C03664=1140.548,355.302,-81.415,-176.440,9.444,148.890
C03665=1140.545,355.549,-81.451,-176.437,9.448,148.890
C03666=1140.541,355.796,-81.486,-176.435,9.451,148.890
C03667=1140.537,356.044,-81.521,-176.433,9.456,148.891
C03668=1140.533,356.292,-81.556,-176.430,9.460,148.891
C03669=1140.529,356.539,-81.592,-176.427,9.464,148.891
C03670=1140.525,356.787,-81.627,-176.425,9.467,148.892
C03671=1140.522,357.034,-81.661,-176.422,9.472,148.892
C03672=1140.518,357.281,-81.697,-176.420,9.476,148.893
C03673=1140.514,357.529,-81.731,-176.417,9.479,148.893
C03674=1140.510,357.776,-81.767,-176.415,9.484,148.893
C03675=1140.506,358.024,-81.803,-176.412,9.488,148.894
C03676=1140.502,358.272,-81.837,-176.409,9.492,148.894
C03677=1140.498,358.519,-81.873,-176.407,9.497,148.894
C03678=1140.494,358.766,-81.908,-176.405,9.500,148.895
C03679=1140.491,359.014,-81.944,-176.402,9.504,148.895
C03680=1140.486,359.262,-81.980,-176.400,9.509,148.896
C03681=1140.482,359.509,-82.014,-176.397,9.513,148.896
C03682=1140.478,359.756,-82.050,-176.395,9.516,148.896
C03683=1140.474,360.004,-82.085,-176.392,9.521,148.897
C03684=1140.471,360.251,-82.121,-176.389,9.525,148.897
C03685=1140.466,360.498,-82.156,-176.387,9.529,148.897
C03686=1140.463,360.746,-82.192,-176.384,9.534,148.898
C03687=1140.459,360.993,-82.227,-176.381,9.538,148.898
C03688=1140.455,361.241,-82.263,-176.379,9.541,148.899
C03689=1140.452,361.488,-82.298,-176.377,9.546,148.899
C03690=1140.447,361.735,-82.333,-176.374,9.550,148.899
C03691=1140.443,361.983,-82.370,-176.371,9.554,148.900
C03692=1140.439,362.230,-82.405,-176.369,9.558,148.900
C03693=1140.436,362.478,-82.441,-176.366,9.563,148.900
C03694=1140.432,362.725,-82.476,-176.364,9.567,148.901
C03695=1140.428,362.973,-82.512,-176.361,9.571,148.901
C03696=1140.425,363.220,-82.547,-176.358,9.575,148.902
C03697=1140.420,363.467,-82.583,-176.356,9.579,148.902
C03698=1140.416,363.715,-82.619,-176.354,9.583,148.902
C03699=1140.412,363.962,-82.654,-176.351,9.587,148.903
C03700=1140.409,364.210,-82.690,-176.348,9.592,148.903
C03701=1140.405,364.457,-82.725,-176.346,9.596,148.904
C03702=1140.400,364.741,-82.767,-176.342,9.601,148.904
C03703=1140.396,365.025,-82.808,-176.340,9.605,148.904
C03704=1140.392,365.309,-82.849,-176.337,9.611,148.905
C03705=1140.387,365.593,-82.890,-176.333,9.616,148.905
C03706=1140.383,365.840,-82.926,-176.331,9.620,148.906
C03707=1140.380,366.087,-82.962,-176.328,9.624,148.906
C03708=1140.375,366.335,-82.998,-176.325,9.629,148.907
C03709=1140.371,366.582,-83.034,-176.323,9.633,148.907
C03710=1140.368,366.830,-83.069,-176.320,9.637,148.907
C03711=1140.364,367.077,-83.106,-176.318,9.642,148.908
C03712=1140.360,367.324,-83.141,-176.315,9.646,148.908
C03713=1140.356,367.572,-83.177,-176.312,9.650,148.909
C03714=1140.352,367.819,-83.214,-176.310,9.654,148.909
C03715=1140.349,368.066,-83.249,-176.307,9.658,148.909
C03716=1140.345,368.314,-83.285,-176.304,9.663,148.910
C03717=1140.341,368.561,-83.322,-176.302,9.667,148.910
C03718=1140.337,368.809,-83.357,-176.299,9.671,148.910
C03719=1140.333,369.056,-83.394,-176.296,9.676,148.911
C03720=1140.329,369.303,-83.430,-176.294,9.680,148.911
C03721=1140.325,369.550,-83.467,-176.291,9.684,148.912
C03722=1140.322,369.798,-83.502,-176.288,9.688,148.912
C03723=1140.318,370.045,-83.539,-176.286,9.692,148.913
C03724=1140.314,370.293,-83.575,-176.284,9.696,148.913
C03725=1140.311,370.540,-83.611,-176.281,9.700,148.913
C03726=1140.306,370.787,-83.647,-176.278,9.705,148.914
C03727=1140.303,371.034,-83.683,-176.276,9.709,148.914
C03728=1140.298,371.282,-83.719,-176.273,9.714,148.915
C03729=1140.295,371.529,-83.756,-176.270,9.718,148.915
C03730=1140.291,371.776,-83.793,-176.268,9.722,148.915
C03731=1140.287,372.024,-83.829,-176.265,9.726,148.916
C03732=1140.283,372.271,-83.865,-176.263,9.731,148.916
C03733=1140.279,372.518,-83.902,-176.260,9.735,148.917
C03734=1140.275,372.766,-83.937,-176.257,9.739,148.917
C03735=1140.271,373.013,-83.974,-176.255,9.744,148.918
C03736=1140.268,373.260,-84.010,-176.253,9.747,148.918
C03737=1140.264,373.508,-84.047,-176.250,9.752,148.918
C03738=1140.260,373.755,-84.084,-176.248,9.756,148.919
C03739=1140.257,374.002,-84.120,-176.245,9.760,148.919
C03740=1140.253,374.249,-84.157,-176.243,9.765,148.920
C03741=1140.249,374.497,-84.193,-176.240,9.768,148.920
C03742=1140.245,374.744,-84.229,-176.238,9.772,148.921
C03743=1140.241,374.991,-84.266,-176.235,9.777,148.921
C03744=1140.237,375.238,-84.302,-176.233,9.781,148.921
C03745=1140.233,375.485,-84.339,-176.231,9.785,148.922
C03746=1140.230,375.734,-84.376,-176.228,9.789,148.922
C03747=1140.226,375.981,-84.412,-176.227,9.793,148.923
C03748=1140.222,376.228,-84.449,-176.224,9.797,148.923
C03749=1140.218,376.475,-84.486,-176.221,9.801,148.924
C03750=1140.215,376.722,-84.522,-176.220,9.805,148.924
C03751=1140.211,376.969,-84.559,-176.217,9.809,148.925
C03752=1140.207,377.217,-84.596,-176.216,9.813,148.925
C03753=1140.203,377.464,-84.633,-176.213,9.818,148.926
C03754=1140.200,377.711,-84.669,-176.211,9.821,148.926
C03755=1140.196,377.958,-84.706,-176.209,9.825,148.926
C03756=1140.191,378.205,-84.743,-176.207,9.829,148.927
C03757=1140.187,378.453,-84.780,-176.205,9.833,148.928
C03758=1140.184,378.701,-84.817,-176.203,9.837,148.928
C03759=1140.180,378.947,-84.853,-176.201,9.841,148.928
C03760=1140.176,379.195,-84.890,-176.199,9.845,148.929
C03761=1140.172,379.442,-84.927,-176.197,9.848,148.929
C03762=1140.168,379.689,-84.964,-176.195,9.852,148.930
C03763=1140.165,379.937,-85.001,-176.194,9.856,148.930
C03764=1140.161,380.184,-85.037,-176.192,9.859,148.931
C03765=1140.157,380.431,-85.074,-176.190,9.863,148.932
C03766=1140.153,380.678,-85.111,-176.188,9.867,148.932
C03767=1140.150,380.925,-85.149,-176.187,9.871,148.933
C03768=1140.146,381.173,-85.186,-176.186,9.874,148.933
C03769=1140.142,381.420,-85.223,-176.184,9.877,148.934
C03770=1140.138,381.667,-85.259,-176.183,9.881,148.934
C03771=1140.135,381.915,-85.296,-176.181,9.885,148.935
C03772=1140.131,382.162,-85.333,-176.180,9.888,148.935
C03773=1140.127,382.408,-85.371,-176.178,9.892,148.936
C03774=1140.123,382.656,-85.408,-176.177,9.895,148.936
C03775=1140.119,382.903,-85.445,-176.176,9.898,148.937
C03776=1140.115,383.151,-85.482,-176.175,9.902,148.937
C03777=1140.112,383.397,-85.519,-176.174,9.905,148.938
C03778=1140.108,383.645,-85.556,-176.173,9.908,148.939
C03779=1140.105,383.892,-85.593,-176.172,9.911,148.939
C03780=1140.101,384.139,-85.630,-176.172,9.914,148.940
C03781=1140.097,384.386,-85.667,-176.171,9.917,148.940
C03782=1140.093,384.634,-85.704,-176.170,9.920,148.941
C03783=1140.089,384.881,-85.741,-176.169,9.924,148.942
C03784=1140.085,385.128,-85.778,-176.168,9.927,148.942
C03785=1140.082,385.375,-85.816,-176.168,9.929,148.943
C03786=1140.078,385.622,-85.853,-176.167,9.932,148.944
C03787=1140.074,385.870,-85.890,-176.167,9.936,148.944
C03788=1140.071,386.117,-85.928,-176.167,9.938,148.945
C03789=1140.067,386.364,-85.965,-176.166,9.941,148.946
C03790=1140.062,386.611,-86.001,-176.166,9.944,148.946
C03791=1140.059,386.859,-86.039,-176.166,9.947,148.947
C03792=1140.055,387.106,-86.076,-176.166,9.949,148.948
C03793=1140.051,387.353,-86.113,-176.166,9.953,148.948
C03794=1140.047,387.600,-86.151,-176.165,9.955,148.949
C03795=1140.044,387.847,-86.188,-176.166,9.957,148.950
C03796=1140.040,388.094,-86.225,-176.166,9.960,148.950
C03797=1140.036,388.341,-86.262,-176.166,9.963,148.951
C03798=1140.032,388.589,-86.300,-176.166,9.965,148.952
C03799=1140.029,388.836,-86.337,-176.166,9.968,148.953
C03800=1140.025,389.083,-86.374,-176.166,9.970,148.953
C03801=1140.021,389.331,-86.411,-176.166,9.973,148.954
C03802=1140.017,389.577,-86.449,-176.167,9.975,148.955
C03803=1140.014,389.825,-86.486,-176.168,9.978,148.955
C03804=1140.010,390.072,-86.524,-176.168,9.980,148.956
C03805=1140.006,390.319,-86.560,-176.169,9.982,148.957
C03806=1140.002,390.606,-86.603,-176.169,9.985,148.958
C03807=1139.998,390.894,-86.647,-176.169,9.988,148.959
C03808=1139.993,391.181,-86.690,-176.170,9.991,148.960
C03809=1139.989,391.468,-86.734,-176.171,9.994,148.961
C03810=1139.986,391.715,-86.771,-176.171,9.996,148.961
C03811=1139.982,391.963,-86.808,-176.173,9.998,148.962
C03812=1139.978,392.209,-86.845,-176.173,10.000,148.963
C03813=1139.974,392.457,-86.882,-176.174,10.002,148.964
C03814=1139.970,392.704,-86.920,-176.174,10.005,148.964
C03815=1139.966,392.951,-86.957,-176.175,10.007,148.965
C03816=1139.963,393.198,-86.995,-176.176,10.009,148.966
C03817=1139.959,393.445,-87.032,-176.177,10.011,148.967
C03818=1139.955,393.693,-87.069,-176.178,10.014,148.968
C03819=1139.951,393.940,-87.107,-176.178,10.016,148.968
C03820=1139.947,394.187,-87.144,-176.179,10.018,148.969
C03821=1139.943,394.434,-87.181,-176.180,10.020,148.970
C03822=1139.940,394.682,-87.219,-176.182,10.022,148.971
C03823=1139.936,394.928,-87.256,-176.183,10.024,148.972
C03824=1139.932,395.176,-87.293,-176.184,10.026,148.972
C03825=1139.928,395.423,-87.330,-176.184,10.029,148.973
C03826=1139.925,395.670,-87.368,-176.185,10.031,148.974
C03827=1139.920,395.917,-87.405,-176.186,10.033,148.975
C03828=1139.917,396.164,-87.443,-176.187,10.035,148.976
C03829=1139.913,396.412,-87.480,-176.188,10.037,148.976
C03830=1139.910,396.659,-87.518,-176.189,10.039,148.977
C03831=1139.906,396.906,-87.554,-176.190,10.041,148.978
C03832=1139.902,397.153,-87.591,-176.192,10.043,148.979
C03833=1139.899,397.401,-87.629,-176.193,10.045,148.980
C03834=1139.895,397.648,-87.666,-176.195,10.046,148.981
C03835=1139.891,397.894,-87.704,-176.196,10.049,148.982
C03836=1139.887,398.142,-87.741,-176.197,10.051,148.982
C03837=1139.883,398.389,-87.778,-176.198,10.053,148.983
C03838=1139.879,398.636,-87.815,-176.199,10.055,148.984
C03839=1139.876,398.883,-87.853,-176.200,10.057,148.985
C03840=1139.872,399.130,-87.890,-176.201,10.059,148.986
C03841=1139.868,399.378,-87.927,-176.202,10.061,148.987
C03842=1139.865,399.625,-87.965,-176.203,10.063,148.987
C03843=1139.861,399.872,-88.002,-176.205,10.065,148.988
C03844=1139.857,400.119,-88.039,-176.206,10.067,148.989
C03845=1139.853,400.367,-88.077,-176.207,10.069,148.990
C03846=1139.850,400.613,-88.114,-176.209,10.071,148.991
C03847=1139.846,400.860,-88.151,-176.210,10.073,148.992
C03848=1139.842,401.108,-88.189,-176.211,10.075,148.992
C03849=1139.838,401.355,-88.226,-176.212,10.077,148.993
C03850=1139.833,401.602,-88.263,-176.213,10.079,148.994
C03851=1139.830,401.850,-88.301,-176.215,10.081,148.995
C03852=1139.826,402.097,-88.338,-176.216,10.083,148.996
C03853=1139.822,402.343,-88.376,-176.217,10.085,148.997
C03854=1139.819,402.591,-88.413,-176.218,10.087,148.998
C03855=1139.815,402.838,-88.450,-176.220,10.089,148.999
C03856=1139.811,403.085,-88.487,-176.221,10.091,148.999
C03857=1139.807,403.333,-88.524,-176.222,10.093,149.000
C03858=1139.804,403.579,-88.562,-176.223,10.095,149.001
C03859=1139.800,403.827,-88.599,-176.225,10.097,149.002
C03860=1139.796,404.074,-88.637,-176.226,10.099,149.003
C03861=1139.792,404.321,-88.674,-176.227,10.101,149.004
C03862=1139.789,404.568,-88.712,-176.228,10.103,149.005
C03863=1139.785,404.816,-88.749,-176.229,10.105,149.005
C03864=1139.781,405.062,-88.786,-176.230,10.107,149.006
C03865=1139.778,405.310,-88.823,-176.232,10.109,149.007
C03866=1139.774,405.557,-88.860,-176.233,10.111,149.008
C03867=1139.770,405.804,-88.898,-176.234,10.114,149.009
C03868=1139.766,406.052,-88.935,-176.236,10.115,149.010
C03869=1139.763,406.298,-88.973,-176.237,10.117,149.010
C03870=1139.759,406.545,-89.009,-176.238,10.119,149.011
C03871=1139.755,406.793,-89.047,-176.239,10.121,149.012
C03872=1139.751,407.040,-89.084,-176.240,10.123,149.013
C03873=1139.747,407.287,-89.121,-176.241,10.125,149.014
C03874=1139.744,407.534,-89.159,-176.242,10.127,149.015
C03875=1139.740,407.782,-89.196,-176.244,10.130,149.016
C03876=1139.736,408.028,-89.233,-176.245,10.132,149.016
C03877=1139.733,408.276,-89.271,-176.246,10.134,149.017
C03878=1139.729,408.523,-89.308,-176.247,10.136,149.018
C03879=1139.725,408.770,-89.345,-176.248,10.138,149.019
C03880=1139.721,409.017,-89.383,-176.249,10.140,149.020
C03881=1139.717,409.264,-89.420,-176.250,10.142,149.021
C03882=1139.714,409.512,-89.457,-176.251,10.144,149.021
C03883=1139.710,409.759,-89.495,-176.252,10.146,149.022
C03884=1139.705,410.006,-89.532,-176.253,10.148,149.023
C03885=1139.702,410.253,-89.570,-176.255,10.150,149.024
C03886=1139.698,410.501,-89.607,-176.256,10.152,149.025
C03887=1139.694,410.747,-89.644,-176.256,10.155,149.026
C03888=1139.691,410.995,-89.682,-176.257,10.157,149.026
C03889=1139.687,411.242,-89.719,-176.258,10.159,149.027
C03890=1139.683,411.489,-89.756,-176.259,10.162,149.028
C03891=1139.679,411.737,-89.793,-176.260,10.164,149.029
C03892=1139.676,411.983,-89.831,-176.261,10.166,149.030
C03893=1139.671,412.230,-89.868,-176.263,10.168,149.031
C03894=1139.668,412.478,-89.906,-176.264,10.170,149.031
C03895=1139.664,412.725,-89.943,-176.264,10.173,149.032
C03896=1139.660,412.972,-89.980,-176.265,10.175,149.033
C03897=1139.657,413.219,-90.017,-176.266,10.177,149.034
C03898=1139.653,413.466,-90.055,-176.267,10.179,149.035
C03899=1139.649,413.713,-90.092,-176.268,10.181,149.035
C03900=1139.646,413.961,-90.129,-176.268,10.184,149.036
C03901=1139.642,414.208,-90.167,-176.269,10.186,149.037
C03902=1139.638,414.455,-90.203,-176.271,10.188,149.038
C03903=1139.634,414.702,-90.241,-176.272,10.190,149.039
C03904=1139.632,414.949,-90.279,-176.272,10.193,149.040
C03905=1139.631,415.196,-90.316,-176.273,10.194,149.040
C03906=1139.630,415.444,-90.353,-176.274,10.196,149.041
C03907=1139.629,415.691,-90.390,-176.275,10.198,149.042
C03908=1139.628,415.938,-90.427,-176.276,10.200,149.043
C03909=1139.630,416.185,-90.464,-176.276,10.203,149.043
C03910=1139.631,416.467,-90.505,-176.277,10.205,149.044
C03911=1139.634,416.749,-90.547,-176.278,10.207,149.045
C03912=1139.637,417.031,-90.589,-176.279,10.210,149.046
C03913=1139.642,417.313,-90.630,-176.280,10.212,149.047
C03914=1139.222,417.315,-90.681,-176.281,10.223,149.050
C03915=1139.217,417.030,-90.639,-176.280,10.221,149.049
C03916=1139.213,416.745,-90.597,-176.280,10.218,149.048
C03917=1139.211,416.459,-90.554,-176.279,10.216,149.048
C03918=1139.209,416.173,-90.513,-176.278,10.214,149.047
C03919=1139.208,415.927,-90.476,-176.277,10.211,149.046
C03920=1139.208,415.679,-90.439,-176.276,10.209,149.045
C03921=1139.209,415.432,-90.401,-176.275,10.208,149.044
C03922=1139.210,415.185,-90.364,-176.275,10.205,149.044
C03923=1139.212,414.937,-90.328,-176.274,10.203,149.043
C03924=1139.214,414.691,-90.290,-176.273,10.201,149.042
C03925=1139.218,414.443,-90.252,-176.272,10.199,149.041
C03926=1139.222,414.196,-90.216,-176.271,10.197,149.040
C03927=1139.225,413.949,-90.178,-176.270,10.194,149.040
C03928=1139.229,413.702,-90.141,-176.269,10.192,149.039
C03929=1139.233,413.455,-90.103,-176.268,10.190,149.038
C03930=1139.236,413.207,-90.066,-176.267,10.188,149.037
C03931=1139.240,412.961,-90.028,-176.267,10.185,149.036
C03932=1139.244,412.713,-89.992,-176.266,10.183,149.035
C03933=1139.247,412.466,-89.954,-176.265,10.181,149.035
C03934=1139.251,412.219,-89.917,-176.264,10.179,149.034
C03935=1139.255,411.972,-89.880,-176.263,10.177,149.033
C03936=1139.259,411.724,-89.842,-176.261,10.174,149.032
C03937=1139.263,411.477,-89.805,-176.260,10.172,149.031
C03938=1139.267,411.231,-89.767,-176.260,10.170,149.030
C03939=1139.270,410.983,-89.730,-176.259,10.167,149.030
C03940=1139.274,410.736,-89.693,-176.258,10.165,149.029
C03941=1139.277,410.488,-89.655,-176.257,10.163,149.028
C03942=1139.281,410.242,-89.618,-176.256,10.161,149.027
C03943=1139.286,409.994,-89.580,-176.255,10.159,149.026
C03944=1139.289,409.747,-89.543,-176.253,10.157,149.025
C03945=1139.293,409.500,-89.506,-176.252,10.155,149.025
C03946=1139.297,409.253,-89.469,-176.251,10.153,149.024
C03947=1139.300,409.005,-89.431,-176.250,10.151,149.023
C03948=1139.305,408.758,-89.394,-176.249,10.149,149.022
C03949=1139.308,408.512,-89.356,-176.248,10.147,149.021
C03950=1139.312,408.264,-89.319,-176.247,10.145,149.020
C03951=1139.316,408.017,-89.282,-176.246,10.143,149.020
C03952=1139.320,407.770,-89.245,-176.244,10.140,149.019
C03953=1139.323,407.523,-89.207,-176.243,10.138,149.018
C03954=1139.327,407.275,-89.170,-176.242,10.136,149.017
C03955=1139.331,407.029,-89.132,-176.241,10.134,149.016
C03956=1139.334,406.781,-89.095,-176.240,10.132,149.015
C03957=1139.338,406.534,-89.058,-176.239,10.130,149.014
C03958=1139.342,406.287,-89.020,-176.238,10.128,149.014
C03959=1139.346,406.039,-88.984,-176.236,10.126,149.013
C03960=1139.349,405.793,-88.946,-176.235,10.123,149.012
C03961=1139.353,405.545,-88.909,-176.234,10.121,149.011
C03962=1139.357,405.298,-88.871,-176.233,10.119,149.010
C03963=1139.361,405.051,-88.834,-176.232,10.117,149.009
C03964=1139.364,404.804,-88.796,-176.231,10.115,149.008
C03965=1139.368,404.557,-88.759,-176.229,10.114,149.007
C03966=1139.372,404.310,-88.722,-176.228,10.112,149.007
C03967=1139.375,404.062,-88.685,-176.227,10.110,149.006
C03968=1139.379,403.815,-88.648,-176.226,10.107,149.005
C03969=1139.384,403.568,-88.610,-176.225,10.105,149.004
C03970=1139.388,403.320,-88.572,-176.223,10.103,149.003
C03971=1139.391,403.074,-88.535,-176.222,10.101,149.002
C03972=1139.395,402.826,-88.498,-176.221,10.099,149.002
C03973=1139.399,402.579,-88.460,-176.219,10.098,149.001
C03974=1139.403,402.332,-88.423,-176.218,10.096,149.000
C03975=1139.406,402.085,-88.385,-176.217,10.093,148.999
C03976=1139.410,401.838,-88.348,-176.216,10.091,148.998
C03977=1139.414,401.591,-88.311,-176.215,10.089,148.997
C03978=1139.417,401.343,-88.274,-176.214,10.087,148.996
C03979=1139.421,401.096,-88.237,-176.212,10.085,148.996
C03980=1139.425,400.849,-88.199,-176.211,10.083,148.995
C03981=1139.429,400.601,-88.162,-176.209,10.081,148.994
C03982=1139.432,400.355,-88.124,-176.208,10.079,148.993
C03983=1139.436,400.108,-88.088,-176.207,10.077,148.992
C03984=1139.440,399.860,-88.050,-176.206,10.075,148.991
C03985=1139.444,399.613,-88.013,-176.205,10.073,148.990
C03986=1139.448,399.367,-87.975,-176.204,10.071,148.990
C03987=1139.451,399.119,-87.938,-176.202,10.069,148.989
C03988=1139.455,398.872,-87.900,-176.201,10.067,148.988
C03989=1139.459,398.625,-87.863,-176.200,10.065,148.987
C03990=1139.462,398.377,-87.826,-176.199,10.063,148.986
C03991=1139.466,398.131,-87.789,-176.197,10.061,148.985
C03992=1139.470,397.883,-87.752,-176.196,10.059,148.984
C03993=1139.473,397.636,-87.714,-176.195,10.057,148.984
C03994=1139.478,397.389,-87.676,-176.194,10.055,148.983
C03995=1139.482,397.141,-87.638,-176.193,10.053,148.982
C03996=1139.486,396.894,-87.602,-176.192,10.051,148.981
C03997=1139.489,396.648,-87.564,-176.191,10.049,148.980
C03998=1139.493,396.400,-87.527,-176.190,10.047,148.980
C03999=1139.497,396.153,-87.489,-176.189,10.045,148.979
C04000=1139.501,395.906,-87.452,-176.188,10.043,148.978
C04001=1139.504,395.658,-87.415,-176.187,10.041,148.977
C04002=1139.508,395.411,-87.378,-176.185,10.038,148.976
C04003=1139.512,395.164,-87.341,-176.184,10.036,148.975
C04004=1139.515,394.917,-87.303,-176.183,10.034,148.975
C04005=1139.519,394.670,-87.266,-176.182,10.032,148.974
C04006=1139.523,394.423,-87.228,-176.182,10.029,148.973
C04007=1139.527,394.175,-87.191,-176.181,10.028,148.972
C04008=1139.531,393.929,-87.154,-176.180,10.026,148.971
C04009=1139.535,393.682,-87.117,-176.179,10.024,148.970
C04010=1139.538,393.434,-87.079,-176.178,10.022,148.970
C04011=1139.542,393.187,-87.042,-176.178,10.019,148.969
C04012=1139.546,392.940,-87.005,-176.177,10.017,148.968
C04013=1139.549,392.693,-86.967,-176.176,10.015,148.967
C04014=1139.553,392.445,-86.930,-176.175,10.013,148.967
C04015=1139.556,392.198,-86.892,-176.174,10.010,148.966
C04016=1139.561,391.951,-86.855,-176.173,10.008,148.965
C04017=1139.564,391.704,-86.818,-176.173,10.006,148.964
C04018=1139.568,391.457,-86.781,-176.172,10.004,148.963
C04019=1139.573,391.169,-86.738,-176.172,10.001,148.963
C04020=1139.577,390.882,-86.694,-176.171,9.998,148.962
C04021=1139.582,390.594,-86.650,-176.170,9.996,148.961
C04022=1139.586,390.307,-86.608,-176.170,9.993,148.960
C04023=1139.589,390.060,-86.570,-176.169,9.990,148.959
C04024=1139.593,389.813,-86.533,-176.169,9.988,148.959
C04025=1139.597,389.566,-86.495,-176.168,9.986,148.958
C04026=1139.601,389.319,-86.458,-176.168,9.983,148.957
C04027=1139.604,389.072,-86.420,-176.168,9.981,148.956
C04028=1139.608,388.824,-86.384,-176.168,9.978,148.956
C04029=1139.612,388.577,-86.347,-176.168,9.975,148.955
C04030=1139.615,388.330,-86.309,-176.168,9.973,148.954
C04031=1139.619,388.083,-86.272,-176.168,9.970,148.954
C04032=1139.623,387.835,-86.235,-176.168,9.968,148.953
C04033=1139.627,387.588,-86.197,-176.168,9.965,148.952
C04034=1139.631,387.341,-86.160,-176.168,9.963,148.951
C04035=1139.635,387.094,-86.123,-176.167,9.960,148.951
C04036=1139.638,386.847,-86.086,-176.167,9.957,148.950
C04037=1139.642,386.599,-86.049,-176.168,9.954,148.949
C04038=1139.646,386.353,-86.011,-176.168,9.952,148.949
C04039=1139.649,386.105,-85.974,-176.168,9.949,148.948
C04040=1139.654,385.858,-85.937,-176.169,9.946,148.947
C04041=1139.657,385.611,-85.899,-176.170,9.943,148.947
C04042=1139.661,385.364,-85.863,-176.170,9.940,148.946
C04043=1139.665,385.116,-85.825,-176.170,9.937,148.946
C04044=1139.669,384.869,-85.788,-176.171,9.934,148.945
C04045=1139.673,384.622,-85.751,-176.171,9.932,148.944
C04046=1139.676,384.374,-85.714,-176.172,9.929,148.944
C04047=1139.680,384.128,-85.676,-176.173,9.925,148.943
C04048=1139.684,383.881,-85.639,-176.174,9.922,148.942
C04049=1139.687,383.633,-85.603,-176.175,9.919,148.942
C04050=1139.691,383.386,-85.566,-176.176,9.915,148.941
C04051=1139.695,383.139,-85.528,-176.177,9.912,148.941
C04052=1139.699,382.892,-85.491,-176.178,9.909,148.940
C04053=1139.702,382.644,-85.454,-176.179,9.906,148.940
C04054=1139.706,382.397,-85.417,-176.180,9.902,148.939
C04055=1139.710,382.150,-85.380,-176.182,9.899,148.939
C04056=1139.714,381.903,-85.342,-176.183,9.895,148.938
C04057=1139.718,381.655,-85.306,-176.185,9.892,148.937
C04058=1139.721,381.408,-85.269,-176.186,9.889,148.937
C04059=1139.725,381.161,-85.232,-176.188,9.885,148.936
C04060=1139.729,380.913,-85.195,-176.189,9.881,148.936
C04061=1139.733,380.667,-85.158,-176.191,9.878,148.935
C04062=1139.737,380.420,-85.121,-176.193,9.874,148.935
C04063=1139.741,380.172,-85.084,-176.194,9.871,148.934
C04064=1139.744,379.925,-85.047,-176.195,9.867,148.934
C04065=1139.748,379.678,-85.010,-176.197,9.863,148.933
C04066=1139.752,379.431,-84.974,-176.199,9.859,148.933
C04067=1139.756,379.183,-84.937,-176.201,9.855,148.932
C04068=1139.760,378.936,-84.900,-176.203,9.852,148.932
C04069=1139.763,378.688,-84.863,-176.205,9.848,148.931
C04070=1139.767,378.441,-84.826,-176.207,9.844,148.931
C04071=1139.771,378.194,-84.790,-176.209,9.840,148.930
C04072=1139.775,377.947,-84.753,-176.211,9.836,148.930
C04073=1139.779,377.700,-84.716,-176.213,9.833,148.930
C04074=1139.783,377.452,-84.679,-176.215,9.828,148.929
C04075=1139.786,377.205,-84.642,-176.217,9.824,148.929
C04076=1139.790,376.958,-84.605,-176.220,9.820,148.928
C04077=1139.794,376.711,-84.569,-176.222,9.817,148.928
C04078=1139.797,376.464,-84.532,-176.224,9.812,148.927
C04079=1139.802,376.217,-84.496,-176.226,9.809,148.927
C04080=1139.805,375.969,-84.458,-176.229,9.804,148.926
C04081=1139.809,375.721,-84.421,-176.231,9.801,148.926
C04082=1139.812,375.475,-84.385,-176.233,9.796,148.925
C04083=1139.817,375.227,-84.348,-176.236,9.792,148.925
C04084=1139.821,374.980,-84.312,-176.237,9.788,148.925
C04085=1139.824,374.733,-84.276,-176.240,9.784,148.924
C04086=1139.828,374.486,-84.239,-176.243,9.780,148.924
C04087=1139.832,374.238,-84.202,-176.245,9.775,148.923
C04088=1139.835,373.991,-84.166,-176.247,9.772,148.923
C04089=1139.840,373.743,-84.129,-176.250,9.768,148.922
C04090=1139.843,373.496,-84.093,-176.252,9.763,148.922
C04091=1139.847,373.249,-84.056,-176.255,9.759,148.922
C04092=1139.851,373.002,-84.019,-176.257,9.754,148.921
C04093=1139.855,372.754,-83.984,-176.260,9.750,148.921
C04094=1139.859,372.507,-83.947,-176.262,9.746,148.920
C04095=1139.862,372.260,-83.911,-176.265,9.742,148.920
C04096=1139.867,372.012,-83.875,-176.267,9.738,148.919
C04097=1139.870,371.765,-83.838,-176.270,9.734,148.919
C04098=1139.874,371.518,-83.801,-176.272,9.729,148.919
C04099=1139.877,371.270,-83.766,-176.275,9.725,148.918
C04100=1139.881,371.023,-83.729,-176.278,9.721,148.918
C04101=1139.885,370.775,-83.693,-176.280,9.716,148.917
C04102=1139.889,370.528,-83.656,-176.283,9.712,148.917
C04103=1139.893,370.281,-83.621,-176.286,9.708,148.917
C04104=1139.897,370.033,-83.584,-176.288,9.704,148.916
C04105=1139.900,369.787,-83.548,-176.291,9.699,148.916
C04106=1139.905,369.539,-83.511,-176.293,9.695,148.915
C04107=1139.908,369.292,-83.475,-176.296,9.691,148.915
C04108=1139.912,369.044,-83.439,-176.299,9.686,148.914
C04109=1139.916,368.797,-83.404,-176.301,9.682,148.914
C04110=1139.920,368.549,-83.367,-176.304,9.678,148.914
C04111=1139.924,368.302,-83.331,-176.307,9.674,148.913
C04112=1139.927,368.055,-83.295,-176.309,9.669,148.913
C04113=1139.932,367.807,-83.259,-176.312,9.665,148.912
C04114=1139.935,367.560,-83.223,-176.315,9.661,148.912
C04115=1139.939,367.312,-83.186,-176.317,9.656,148.912
C04116=1139.944,367.066,-83.151,-176.320,9.652,148.911
C04117=1139.947,366.818,-83.116,-176.323,9.648,148.911
C04118=1139.951,366.571,-83.079,-176.325,9.643,148.910
C04119=1139.955,366.324,-83.043,-176.328,9.639,148.910
C04120=1139.959,366.076,-83.008,-176.331,9.635,148.910
C04121=1139.963,365.829,-82.971,-176.333,9.631,148.909
C04122=1139.966,365.581,-82.935,-176.336,9.626,148.909
C04123=1139.971,365.298,-82.894,-176.338,9.622,148.908
C04124=1139.975,365.014,-82.853,-176.342,9.617,148.908
C04125=1139.980,364.730,-82.812,-176.345,9.612,148.907
C04126=1139.984,364.446,-82.771,-176.347,9.607,148.907
C04127=1139.987,364.199,-82.735,-176.350,9.603,148.907
C04128=1139.992,363.951,-82.699,-176.353,9.599,148.906
C04129=1139.996,363.704,-82.664,-176.355,9.595,148.906
C04130=1140.000,363.456,-82.628,-176.358,9.590,148.905
C04131=1140.003,363.209,-82.593,-176.361,9.586,148.905
C04132=1140.007,362.961,-82.557,-176.363,9.582,148.905
C04133=1140.011,362.714,-82.521,-176.366,9.577,148.904
C04134=1140.015,362.466,-82.486,-176.369,9.573,148.904
C04135=1140.019,362.219,-82.450,-176.371,9.569,148.903
C04136=1140.023,361.972,-82.415,-176.373,9.565,148.903
C04137=1140.027,361.724,-82.379,-176.376,9.561,148.903
C04138=1140.030,361.477,-82.344,-176.379,9.557,148.902
C04139=1140.035,361.229,-82.308,-176.381,9.552,148.902
C04140=1140.038,360.982,-82.272,-176.384,9.548,148.902
C04141=1140.043,360.735,-82.237,-176.387,9.544,148.901
C04142=1140.046,360.487,-82.201,-176.389,9.540,148.901
C04143=1140.050,360.240,-82.166,-176.391,9.536,148.901
C04144=1140.054,359.992,-82.130,-176.394,9.532,148.900
C04145=1140.057,359.745,-82.095,-176.396,9.528,148.900
C04146=1140.061,359.498,-82.060,-176.399,9.524,148.899
C04147=1140.065,359.250,-82.024,-176.402,9.519,148.899
C04148=1140.069,359.002,-81.989,-176.404,9.516,148.899
C04149=1140.073,358.755,-81.954,-176.407,9.512,148.898
C04150=1140.077,358.508,-81.918,-176.409,9.507,148.898
C04151=1140.081,358.261,-81.883,-176.412,9.503,148.897
C04152=1140.084,358.013,-81.847,-176.415,9.499,148.897
C04153=1140.088,357.765,-81.812,-176.417,9.495,148.897
C04154=1140.093,357.518,-81.777,-176.420,9.491,148.896
C04155=1140.096,357.271,-81.742,-176.422,9.487,148.896
C04156=1140.100,357.022,-81.707,-176.425,9.482,148.895
C04157=1140.104,356.775,-81.671,-176.427,9.479,148.895
C04158=1140.108,356.528,-81.636,-176.429,9.475,148.895
C04159=1140.112,356.280,-81.601,-176.432,9.470,148.894
C04160=1140.116,356.033,-81.566,-176.435,9.466,148.894
C04161=1140.120,355.786,-81.531,-176.437,9.463,148.894
C04162=1140.124,355.538,-81.496,-176.439,9.458,148.893
C04163=1140.128,355.290,-81.460,-176.442,9.454,148.893
C04164=1140.132,355.043,-81.425,-176.445,9.450,148.893
C04165=1140.136,354.795,-81.390,-176.447,9.447,148.892
C04166=1140.140,354.548,-81.355,-176.450,9.442,148.892
C04167=1140.143,354.301,-81.321,-176.452,9.438,148.891
C04168=1140.147,354.053,-81.285,-176.454,9.434,148.891
C04169=1140.151,353.805,-81.250,-176.457,9.430,148.891
C04170=1140.155,353.558,-81.215,-176.460,9.426,148.890
C04171=1140.159,353.310,-81.180,-176.462,9.422,148.890
C04172=1140.163,353.063,-81.145,-176.464,9.418,148.890
C04173=1140.168,352.815,-81.110,-176.467,9.414,148.889
C04174=1140.170,352.568,-81.075,-176.470,9.410,148.889
C04175=1140.175,352.321,-81.041,-176.473,9.406,148.889
C04176=1140.179,352.072,-81.006,-176.475,9.402,148.888
C04177=1140.183,351.825,-80.971,-176.478,9.398,148.888
C04178=1140.187,351.577,-80.936,-176.480,9.394,148.888
C04179=1140.190,351.330,-80.902,-176.482,9.390,148.887
C04180=1140.195,351.083,-80.867,-176.485,9.386,148.887
C04181=1140.199,350.835,-80.832,-176.487,9.381,148.886
C04182=1140.203,350.587,-80.797,-176.490,9.378,148.886
C04183=1140.206,350.340,-80.762,-176.492,9.374,148.886
C04184=1140.210,350.092,-80.728,-176.495,9.370,148.886
C04185=1140.215,349.845,-80.693,-176.498,9.365,148.885
C04186=1140.219,349.596,-80.658,-176.500,9.362,148.885
C04187=1140.222,349.350,-80.624,-176.503,9.358,148.884
C04188=1140.226,349.102,-80.589,-176.505,9.354,148.884
C04189=1140.231,348.854,-80.554,-176.507,9.350,148.884
C04190=1140.234,348.607,-80.520,-176.510,9.346,148.884
C04191=1140.238,348.360,-80.485,-176.513,9.342,148.883
C04192=1140.242,348.112,-80.450,-176.515,9.338,148.883
C04193=1140.246,347.865,-80.416,-176.518,9.334,148.882
C04194=1140.250,347.617,-80.381,-176.521,9.330,148.882
C04195=1140.255,347.369,-80.347,-176.523,9.326,148.882
C04196=1140.258,347.121,-80.313,-176.525,9.322,148.882
C04197=1140.262,346.874,-80.278,-176.528,9.318,148.881
C04198=1140.266,346.626,-80.244,-176.530,9.315,148.881
C04199=1140.270,346.379,-80.210,-176.533,9.310,148.880
C04200=1140.274,346.130,-80.175,-176.536,9.306,148.880
C04201=1140.278,345.883,-80.141,-176.538,9.303,148.880
C04202=1140.282,345.635,-80.106,-176.541,9.298,148.880
C04203=1140.286,345.388,-80.072,-176.543,9.294,148.879
C04204=1140.290,345.141,-80.038,-176.545,9.291,148.879
C04205=1140.294,344.893,-80.003,-176.548,9.287,148.879
C04206=1140.298,344.646,-79.969,-176.551,9.282,148.878
C04207=1140.301,344.398,-79.935,-176.553,9.279,148.878
C04208=1140.306,344.150,-79.900,-176.556,9.275,148.878
C04209=1140.309,343.902,-79.866,-176.559,9.271,148.877
C04210=1140.314,343.655,-79.832,-176.561,9.267,148.877
C04211=1140.318,343.408,-79.798,-176.563,9.263,148.877
C04212=1140.322,343.160,-79.763,-176.566,9.259,148.876
C04213=1140.326,342.912,-79.730,-176.568,9.255,148.876
C04214=1140.330,342.665,-79.695,-176.571,9.251,148.876
C04215=1140.333,342.417,-79.661,-176.574,9.247,148.875
C04216=1140.338,342.169,-79.627,-176.576,9.244,148.875
C04217=1140.341,341.922,-79.592,-176.579,9.240,148.875
C04218=1140.346,341.674,-79.559,-176.582,9.235,148.874
C04219=1140.350,341.426,-79.525,-176.584,9.232,148.874
C04220=1140.353,341.179,-79.490,-176.586,9.228,148.874
C04221=1140.358,340.931,-79.456,-176.589,9.224,148.874
C04222=1140.362,340.684,-79.423,-176.592,9.220,148.873
C04223=1140.366,340.435,-79.388,-176.594,9.216,148.873
C04224=1140.370,340.188,-79.354,-176.596,9.213,148.873
C04225=1140.374,339.941,-79.321,-176.599,9.208,148.872
C04226=1140.378,339.692,-79.286,-176.602,9.204,148.872
C04227=1140.383,339.412,-79.248,-176.605,9.200,148.872
C04228=1140.387,339.132,-79.210,-176.607,9.196,148.871
C04229=1140.391,338.851,-79.171,-176.610,9.192,148.871
C04230=1140.396,338.570,-79.133,-176.613,9.187,148.871
C04231=1140.400,338.323,-79.100,-176.616,9.183,148.870
C04232=1140.405,338.075,-79.065,-176.619,9.179,148.870
C04233=1140.408,337.827,-79.031,-176.621,9.176,148.870
C04234=1140.412,337.580,-78.998,-176.623,9.171,148.869
C04235=1140.416,337.333,-78.964,-176.626,9.167,148.869
C04236=1140.420,337.084,-78.930,-176.629,9.164,148.869
C04237=1140.424,336.837,-78.896,-176.631,9.160,148.869
C04238=1140.428,336.589,-78.863,-176.634,9.156,148.868
C04239=1140.432,336.341,-78.830,-176.636,9.152,148.868
C04240=1140.436,336.093,-78.795,-176.639,9.148,148.868
C04241=1140.440,335.845,-78.762,-176.641,9.145,148.868
C04242=1140.444,335.598,-78.728,-176.644,9.141,148.867
C04243=1140.448,335.351,-78.695,-176.647,9.137,148.867
C04244=1140.453,335.103,-78.661,-176.649,9.133,148.867
C04245=1140.456,334.855,-78.627,-176.652,9.129,148.866
C04246=1140.460,334.607,-78.594,-176.654,9.126,148.866
C04247=1140.464,334.360,-78.560,-176.657,9.122,148.866
C04248=1140.469,334.112,-78.526,-176.659,9.118,148.866
C04249=1140.473,333.864,-78.493,-176.662,9.114,148.865
C04250=1140.476,333.616,-78.460,-176.664,9.111,148.865
C04251=1140.480,333.369,-78.426,-176.667,9.107,148.865
C04252=1140.484,333.121,-78.393,-176.670,9.102,148.864
C04253=1140.488,332.873,-78.360,-176.672,9.099,148.864
C04254=1140.493,332.626,-78.326,-176.675,9.095,148.864
C04255=1140.496,332.379,-78.293,-176.677,9.092,148.864
C04256=1140.500,332.130,-78.259,-176.680,9.087,148.863
C04257=1140.504,331.882,-78.226,-176.682,9.084,148.863
C04258=1140.508,331.635,-78.193,-176.685,9.080,148.863
C04259=1140.513,331.387,-78.159,-176.688,9.076,148.863
C04260=1140.517,331.139,-78.126,-176.691,9.073,148.863
C04261=1140.521,330.892,-78.092,-176.693,9.068,148.862
C04262=1140.525,330.644,-78.059,-176.695,9.065,148.862
C04263=1140.529,330.396,-78.025,-176.698,9.061,148.862
C04264=1140.533,330.148,-77.992,-176.701,9.058,148.861
C04265=1140.537,329.900,-77.959,-176.704,9.053,148.861
C04266=1140.540,329.653,-77.926,-176.705,9.050,148.861
C04267=1140.545,329.405,-77.893,-176.708,9.046,148.861
C04268=1140.549,329.157,-77.860,-176.711,9.042,148.860
C04269=1140.553,328.910,-77.827,-176.714,9.038,148.860
C04270=1140.557,328.662,-77.794,-176.717,9.034,148.860
C04271=1140.561,328.414,-77.761,-176.719,9.031,148.860
C04272=1140.565,328.166,-77.727,-176.721,9.027,148.859
C04273=1140.569,327.919,-77.694,-176.724,9.023,148.859
C04274=1140.573,327.671,-77.661,-176.727,9.019,148.859
C04275=1140.578,327.423,-77.628,-176.729,9.016,148.859
C04276=1140.582,327.175,-77.595,-176.732,9.012,148.858
C04277=1140.586,326.927,-77.562,-176.734,9.009,148.858
C04278=1140.590,326.680,-77.530,-176.737,9.005,148.858
C04279=1140.594,326.432,-77.497,-176.739,9.001,148.858
C04280=1140.598,326.184,-77.464,-176.742,8.997,148.857
C04281=1140.602,325.936,-77.430,-176.745,8.993,148.857
C04282=1140.606,325.689,-77.397,-176.747,8.990,148.857
C04283=1140.611,325.440,-77.365,-176.750,8.986,148.857
C04284=1140.614,325.193,-77.332,-176.753,8.982,148.857
C04285=1140.618,324.945,-77.299,-176.756,8.978,148.856
C04286=1140.622,324.698,-77.266,-176.758,8.975,148.856
C04287=1140.627,324.449,-77.233,-176.761,8.971,148.856
C04288=1140.630,324.202,-77.201,-176.763,8.968,148.856
C04289=1140.634,323.954,-77.168,-176.766,8.963,148.855
C04290=1140.638,323.706,-77.135,-176.768,8.960,148.855
C04291=1140.643,323.458,-77.102,-176.771,8.956,148.855
C04292=1140.646,323.211,-77.070,-176.773,8.953,148.855
C04293=1140.650,322.963,-77.036,-176.776,8.949,148.854
C04294=1140.655,322.714,-77.004,-176.778,8.945,148.854
C04295=1140.658,322.467,-76.971,-176.781,8.941,148.854
C04296=1140.662,322.219,-76.938,-176.784,8.938,148.854
C04297=1140.667,321.971,-76.906,-176.787,8.934,148.854
C04298=1140.670,321.724,-76.873,-176.789,8.931,148.853
C04299=1140.675,321.475,-76.841,-176.792,8.927,148.853
C04300=1140.679,321.227,-76.808,-176.794,8.923,148.853
C04301=1140.683,320.979,-76.776,-176.797,8.919,148.853
C04302=1140.687,320.732,-76.743,-176.800,8.916,148.853
C04303=1140.692,320.484,-76.711,-176.802,8.912,148.852
C04304=1140.695,320.237,-76.678,-176.805,8.909,148.852
C04305=1140.700,319.988,-76.646,-176.808,8.905,148.852
C04306=1140.703,319.741,-76.613,-176.810,8.901,148.852
C04307=1140.707,319.493,-76.581,-176.813,8.897,148.852
C04308=1140.712,319.245,-76.547,-176.815,8.894,148.851
C04309=1140.715,318.997,-76.516,-176.818,8.890,148.851
C04310=1140.720,318.748,-76.483,-176.821,8.887,148.851
C04311=1140.724,318.502,-76.451,-176.823,8.884,148.851
C04312=1140.728,318.253,-76.419,-176.826,8.879,148.851
C04313=1140.732,318.006,-76.386,-176.828,8.876,148.850
C04314=1140.736,317.758,-76.354,-176.831,8.872,148.850
C04315=1140.740,317.510,-76.322,-176.833,8.869,148.850
C04316=1140.744,317.262,-76.289,-176.836,8.865,148.850
C04317=1140.748,317.014,-76.257,-176.839,8.862,148.850
C04318=1140.753,316.766,-76.225,-176.842,8.857,148.849
C04319=1140.756,316.518,-76.193,-176.844,8.854,148.849
C04320=1140.760,316.270,-76.160,-176.847,8.850,148.849
C04321=1140.764,316.022,-76.128,-176.849,8.847,148.849
C04322=1140.769,315.775,-76.096,-176.852,8.843,148.848
C04323=1140.773,315.527,-76.064,-176.855,8.840,148.848
C04324=1140.777,315.279,-76.031,-176.857,8.836,148.848
C04325=1140.781,315.031,-75.999,-176.860,8.832,148.848
C04326=1140.785,314.784,-75.967,-176.862,8.829,148.848
C04327=1140.789,314.535,-75.935,-176.865,8.825,148.847
C04328=1140.793,314.287,-75.903,-176.868,8.822,148.848
C04329=1140.798,314.039,-75.871,-176.871,8.818,148.847
C04330=1140.802,313.791,-75.839,-176.873,8.815,148.847
C04331=1140.806,313.513,-75.803,-176.876,8.811,148.847
C04332=1140.811,313.235,-75.767,-176.879,8.806,148.847
C04333=1140.815,312.958,-75.731,-176.882,8.802,148.846
C04334=1140.820,312.680,-75.695,-176.885,8.798,148.846
C04335=1140.824,312.432,-75.663,-176.887,8.795,148.846
C04336=1140.829,312.184,-75.631,-176.890,8.791,148.846
C04337=1140.833,311.936,-75.599,-176.893,8.788,148.846
C04338=1140.836,311.688,-75.568,-176.896,8.784,148.846
C04339=1140.840,311.440,-75.536,-176.898,8.781,148.845
C04340=1140.845,311.193,-75.504,-176.901,8.777,148.845
C04341=1140.849,310.944,-75.472,-176.903,8.773,148.845
C04342=1140.852,310.696,-75.440,-176.906,8.770,148.845
C04343=1140.857,310.449,-75.408,-176.909,8.766,148.845
C04344=1140.861,310.201,-75.376,-176.911,8.763,148.845
C04345=1140.866,309.953,-75.345,-176.914,8.759,148.844
C04346=1140.869,309.705,-75.313,-176.917,8.756,148.844
C04347=1140.873,309.457,-75.282,-176.919,8.752,148.844
C04348=1140.878,309.209,-75.249,-176.922,8.748,148.844
C04349=1140.882,308.961,-75.218,-176.924,8.745,148.844
C04350=1140.886,308.713,-75.186,-176.927,8.741,148.843
C04351=1140.890,308.465,-75.155,-176.930,8.738,148.843
C04352=1140.894,308.217,-75.123,-176.933,8.734,148.843
C04353=1140.899,307.969,-75.091,-176.935,8.731,148.843
C04354=1140.903,307.721,-75.059,-176.938,8.728,148.843
C04355=1140.907,307.473,-75.028,-176.941,8.723,148.843
C04356=1140.911,307.225,-74.997,-176.943,8.721,148.843
C04357=1140.915,306.977,-74.965,-176.946,8.717,148.843
C04358=1140.919,306.730,-74.933,-176.949,8.713,148.842
C04359=1140.924,306.481,-74.902,-176.951,8.710,148.842
C04360=1140.928,306.234,-74.870,-176.954,8.706,148.842
C04361=1140.932,305.986,-74.838,-176.957,8.703,148.842
C04362=1140.936,305.737,-74.807,-176.959,8.700,148.842
C04363=1140.940,305.490,-74.776,-176.962,8.696,148.842
C04364=1140.944,305.241,-74.745,-176.964,8.692,148.841
C04365=1140.948,304.994,-74.713,-176.968,8.689,148.841
C04366=1140.952,304.746,-74.681,-176.970,8.685,148.841
C04367=1140.957,304.498,-74.650,-176.972,8.682,148.841
C04368=1140.960,304.250,-74.619,-176.975,8.678,148.841
C04369=1140.965,304.002,-74.588,-176.978,8.675,148.841
C04370=1140.969,303.754,-74.556,-176.980,8.672,148.841
C04371=1140.973,303.506,-74.525,-176.983,8.668,148.840
C04372=1140.977,303.258,-74.493,-176.986,8.664,148.840
C04373=1140.982,303.010,-74.463,-176.989,8.661,148.840
C04374=1140.985,302.762,-74.431,-176.991,8.657,148.840
C04375=1140.990,302.514,-74.400,-176.994,8.654,148.840
C04376=1140.994,302.266,-74.368,-176.997,8.650,148.840
C04377=1140.998,302.018,-74.337,-176.999,8.647,148.840
C04378=1141.002,301.769,-74.306,-177.002,8.644,148.840
C04379=1141.007,301.522,-74.275,-177.005,8.640,148.839
C04380=1141.011,301.274,-74.244,-177.007,8.637,148.839
C04381=1141.015,301.025,-74.213,-177.010,8.634,148.839
C04382=1141.020,300.778,-74.181,-177.013,8.630,148.839
C04383=1141.024,300.529,-74.150,-177.015,8.626,148.839
C04384=1141.028,300.281,-74.120,-177.018,8.623,148.839
C04385=1141.032,300.033,-74.088,-177.021,8.619,148.839
C04386=1141.036,299.785,-74.058,-177.023,8.616,148.838
C04387=1141.040,299.537,-74.027,-177.026,8.613,148.839
C04388=1141.044,299.289,-73.995,-177.029,8.609,148.838
C04389=1141.049,299.041,-73.964,-177.031,8.606,148.838
C04390=1141.053,298.793,-73.933,-177.034,8.602,148.838
C04391=1141.057,298.545,-73.902,-177.037,8.599,148.838
C04392=1141.061,298.298,-73.871,-177.039,8.596,148.838
C04393=1141.065,298.049,-73.840,-177.042,8.592,148.838
C04394=1141.070,297.801,-73.809,-177.045,8.589,148.838
C04395=1141.074,297.552,-73.778,-177.047,8.585,148.837
C04396=1141.078,297.305,-73.748,-177.050,8.582,148.837
C04397=1141.082,297.057,-73.717,-177.053,8.578,148.837
C04398=1141.086,296.808,-73.686,-177.055,8.575,148.837
C04399=1141.090,296.561,-73.655,-177.058,8.572,148.837
C04400=1141.095,296.313,-73.624,-177.061,8.568,148.837
C04401=1141.098,296.065,-73.594,-177.063,8.565,148.837
C04402=1141.103,295.817,-73.563,-177.066,8.562,148.837
C04403=1141.107,295.569,-73.532,-177.069,8.558,148.837
C04404=1141.111,295.320,-73.501,-177.072,8.555,148.837
C04405=1141.115,295.072,-73.471,-177.074,8.552,148.836
C04406=1141.120,294.824,-73.440,-177.077,8.547,148.836
C04407=1141.123,294.576,-73.409,-177.080,8.545,148.836
C04408=1141.128,294.328,-73.379,-177.082,8.541,148.836
C04409=1141.133,294.080,-73.348,-177.085,8.538,148.836
C04410=1141.136,293.832,-73.317,-177.088,8.534,148.836
C04411=1141.140,293.584,-73.287,-177.090,8.531,148.836
C04412=1141.145,293.336,-73.256,-177.093,8.528,148.836
C04413=1141.149,293.088,-73.226,-177.096,8.524,148.836
C04414=1141.153,292.839,-73.195,-177.099,8.521,148.836
C04415=1141.157,292.591,-73.165,-177.101,8.518,148.835
C04416=1141.162,292.343,-73.134,-177.104,8.514,148.835
C04417=1141.166,292.095,-73.104,-177.107,8.511,148.835
C04418=1141.170,291.847,-73.073,-177.109,8.508,148.835
C04419=1141.174,291.599,-73.042,-177.112,8.504,148.835
C04420=1141.178,291.351,-73.013,-177.115,8.501,148.835
C04421=1141.183,291.103,-72.982,-177.117,8.498,148.835
C04422=1141.186,290.854,-72.951,-177.120,8.494,148.835
C04423=1141.191,290.607,-72.921,-177.123,8.491,148.835
C04424=1141.195,290.359,-72.891,-177.126,8.487,148.835
C04425=1141.200,290.110,-72.860,-177.128,8.484,148.834
C04426=1141.204,289.863,-72.830,-177.131,8.480,148.834
C04427=1141.208,289.614,-72.799,-177.134,8.477,148.834
C04428=1141.212,289.366,-72.770,-177.136,8.474,148.834
C04429=1141.216,289.118,-72.739,-177.139,8.471,148.834
C04430=1141.220,288.870,-72.709,-177.142,8.467,148.834
C04431=1141.225,288.622,-72.679,-177.144,8.464,148.834
C04432=1141.228,288.373,-72.648,-177.147,8.461,148.834
C04433=1141.233,288.125,-72.617,-177.149,8.458,148.834
C04434=1141.237,287.877,-72.588,-177.153,8.454,148.834
C04435=1141.243,287.602,-72.554,-177.155,8.451,148.834
C04436=1141.247,287.326,-72.520,-177.159,8.447,148.834
C04437=1141.251,287.050,-72.487,-177.161,8.443,148.834
C04438=1141.256,286.775,-72.454,-177.165,8.439,148.834
C04439=1141.261,286.527,-72.424,-177.167,8.436,148.833
C04440=1141.264,286.279,-72.394,-177.170,8.433,148.833
C04441=1141.269,286.031,-72.364,-177.172,8.430,148.833
C04442=1141.273,285.782,-72.333,-177.176,8.426,148.833
C04443=1141.277,285.534,-72.304,-177.178,8.423,148.833
C04444=1141.281,285.286,-72.273,-177.181,8.420,148.833
C04445=1141.286,285.038,-72.244,-177.184,8.417,148.833
C04446=1141.289,284.790,-72.213,-177.187,8.413,148.833
C04447=1141.294,284.542,-72.183,-177.189,8.410,148.833
C04448=1141.299,284.293,-72.154,-177.192,8.407,148.833
C04449=1141.302,284.046,-72.124,-177.194,8.404,148.833
C04450=1141.307,283.797,-72.094,-177.197,8.400,148.833
C04451=1141.312,283.549,-72.064,-177.200,8.397,148.833
C04452=1141.315,283.301,-72.034,-177.202,8.393,148.833
C04453=1141.320,283.053,-72.005,-177.205,8.390,148.833
C04454=1141.325,282.804,-71.975,-177.208,8.387,148.833
C04455=1141.328,282.557,-71.944,-177.211,8.383,148.833
C04456=1141.333,282.309,-71.915,-177.214,8.380,148.833
C04457=1141.337,282.060,-71.886,-177.216,8.377,148.832
C04458=1141.341,281.812,-71.855,-177.219,8.374,148.832
C04459=1141.346,281.564,-71.825,-177.222,8.370,148.832
C04460=1141.350,281.316,-71.796,-177.225,8.367,148.832
C04461=1141.354,281.068,-71.766,-177.227,8.364,148.832
C04462=1141.358,280.819,-71.737,-177.230,8.361,148.832
C04463=1141.363,280.571,-71.706,-177.232,8.358,148.832
C04464=1141.367,280.323,-71.677,-177.235,8.354,148.832
C04465=1141.371,280.075,-71.647,-177.238,8.351,148.832
C04466=1141.375,279.826,-71.618,-177.241,8.348,148.832
C04467=1141.379,279.578,-71.588,-177.243,8.345,148.832
C04468=1141.384,279.330,-71.559,-177.246,8.342,148.832
C04469=1141.388,279.082,-71.529,-177.249,8.338,148.832
C04470=1141.392,278.834,-71.499,-177.252,8.335,148.832
C04471=1141.397,278.585,-71.469,-177.254,8.332,148.832
C04472=1141.401,278.337,-71.440,-177.257,8.329,148.832
C04473=1141.405,278.089,-71.410,-177.260,8.325,148.832
C04474=1141.409,277.841,-71.381,-177.263,8.322,148.832
C04475=1141.413,277.592,-71.351,-177.265,8.319,148.832
C04476=1141.417,277.344,-71.322,-177.268,8.316,148.832
C04477=1141.422,277.096,-71.293,-177.271,8.313,148.832
C04478=1141.426,276.848,-71.263,-177.273,8.310,148.832
C04479=1141.430,276.599,-71.234,-177.276,8.306,148.831
C04480=1141.434,276.351,-71.204,-177.279,8.303,148.831
C04481=1141.439,276.103,-71.175,-177.282,8.300,148.832
C04482=1141.443,275.855,-71.146,-177.284,8.297,148.831
C04483=1141.448,275.606,-71.117,-177.287,8.294,148.831
C04484=1141.452,275.358,-71.087,-177.290,8.290,148.831
C04485=1141.456,275.110,-71.058,-177.293,8.287,148.831
C04486=1141.460,274.862,-71.029,-177.295,8.284,148.831
C04487=1141.464,274.613,-70.999,-177.298,8.281,148.831
C04488=1141.469,274.365,-70.970,-177.301,8.278,148.831
C04489=1141.473,274.117,-70.941,-177.303,8.275,148.831
C04490=1141.478,273.869,-70.912,-177.307,8.271,148.831
C04491=1141.481,273.621,-70.883,-177.309,8.268,148.831
C04492=1141.485,273.372,-70.854,-177.312,8.265,148.831
C04493=1141.490,273.124,-70.824,-177.315,8.262,148.831
C04494=1141.494,272.876,-70.795,-177.317,8.259,148.831
C04495=1141.499,272.628,-70.766,-177.320,8.256,148.831
C04496=1141.503,272.379,-70.737,-177.323,8.252,148.831
C04497=1141.507,272.131,-70.707,-177.325,8.249,148.831
C04498=1141.512,271.882,-70.679,-177.328,8.246,148.831
C04499=1141.515,271.634,-70.650,-177.331,8.243,148.831
C04500=1141.520,271.387,-70.621,-177.333,8.240,148.831
C04501=1141.524,271.138,-70.592,-177.336,8.237,148.831
C04502=1141.529,270.889,-70.562,-177.340,8.233,148.831
C04503=1141.533,270.641,-70.533,-177.342,8.230,148.831
C04504=1141.537,270.393,-70.505,-177.345,8.227,148.831
C04505=1141.541,270.145,-70.476,-177.347,8.224,148.831
C04506=1141.546,269.896,-70.447,-177.350,8.221,148.831
C04507=1141.550,269.648,-70.418,-177.353,8.218,148.831
C04508=1141.554,269.400,-70.388,-177.355,8.215,148.831
C04509=1141.559,269.152,-70.360,-177.359,8.211,148.831
C04510=1141.563,268.904,-70.331,-177.362,8.208,148.831
C04511=1141.567,268.655,-70.302,-177.364,8.205,148.831
C04512=1141.572,268.407,-70.273,-177.367,8.202,148.831
C04513=1141.576,268.158,-70.245,-177.369,8.199,148.831
C04514=1141.580,267.910,-70.215,-177.372,8.196,148.831
C04515=1141.584,267.661,-70.187,-177.375,8.193,148.831
C04516=1141.588,267.414,-70.158,-177.378,8.189,148.831
C04517=1141.593,267.165,-70.129,-177.381,8.186,148.831
C04518=1141.597,266.916,-70.101,-177.383,8.183,148.831
C04519=1141.602,266.669,-70.072,-177.386,8.180,148.831
C04520=1141.606,266.420,-70.044,-177.389,8.177,148.831
C04521=1141.610,266.172,-70.014,-177.391,8.174,148.831
C04522=1141.615,265.924,-69.986,-177.394,8.171,148.831
C04523=1141.619,265.675,-69.958,-177.397,8.168,148.831
C04524=1141.623,265.427,-69.928,-177.399,8.165,148.831
C04525=1141.628,265.179,-69.900,-177.403,8.161,148.831
C04526=1141.632,264.930,-69.872,-177.406,8.158,148.831
C04527=1141.636,264.682,-69.844,-177.408,8.155,148.831
C04528=1141.641,264.434,-69.814,-177.411,8.152,148.831
C04529=1141.645,264.185,-69.786,-177.413,8.149,148.831
C04530=1141.649,263.937,-69.758,-177.416,8.146,148.831
C04531=1141.654,263.688,-69.729,-177.419,8.143,148.831
C04532=1141.657,263.440,-69.700,-177.421,8.140,148.831
C04533=1141.662,263.192,-69.672,-177.424,8.137,148.831
C04534=1141.666,262.944,-69.644,-177.428,8.133,148.831
C04535=1141.671,262.695,-69.615,-177.430,8.130,148.831
C04536=1141.675,262.447,-69.587,-177.433,8.127,148.831
C04537=1141.679,262.199,-69.558,-177.435,8.124,148.831
C04538=1141.684,261.951,-69.530,-177.438,8.121,148.831
C04539=1141.689,261.677,-69.499,-177.441,8.118,148.831
C04540=1141.693,261.403,-69.468,-177.444,8.115,148.831
C04541=1141.698,261.129,-69.436,-177.447,8.112,148.831
C04542=1141.703,260.857,-69.405,-177.451,8.108,148.831
C04543=1141.707,260.608,-69.376,-177.453,8.105,148.831
C04544=1141.712,260.360,-69.348,-177.456,8.102,148.831
C04545=1141.715,260.111,-69.320,-177.458,8.099,148.831
C04546=1141.720,259.863,-69.292,-177.461,8.096,148.831
C04547=1141.724,259.615,-69.264,-177.464,8.093,148.831
C04548=1141.729,259.366,-69.235,-177.467,8.090,148.831
C04549=1141.733,259.118,-69.207,-177.470,8.086,148.831
C04550=1141.737,258.870,-69.180,-177.473,8.083,148.831
C04551=1141.742,258.621,-69.151,-177.475,8.080,148.831
C04552=1141.746,258.373,-69.123,-177.478,8.077,148.832
C04553=1141.751,258.124,-69.094,-177.481,8.074,148.832
C04554=1141.755,257.876,-69.067,-177.484,8.071,148.832
C04555=1141.759,257.627,-69.039,-177.486,8.068,148.832
C04556=1141.764,257.379,-69.011,-177.489,8.065,148.832
C04557=1141.768,257.130,-68.983,-177.492,8.062,148.832
C04558=1141.772,256.883,-68.955,-177.494,8.059,148.832
C04559=1141.777,256.634,-68.926,-177.497,8.056,148.832
C04560=1141.781,256.386,-68.898,-177.500,8.054,148.832
C04561=1141.785,256.137,-68.870,-177.503,8.051,148.832
C04562=1141.790,255.889,-68.843,-177.506,8.048,148.832
C04563=1141.794,255.640,-68.814,-177.508,8.044,148.832
C04564=1141.798,255.392,-68.787,-177.511,8.042,148.832
C04565=1141.803,255.144,-68.759,-177.514,8.038,148.832
C04566=1141.807,254.895,-68.731,-177.517,8.035,148.832
C04567=1141.812,254.647,-68.703,-177.520,8.032,148.832
C04568=1141.816,254.398,-68.675,-177.522,8.029,148.832
C04569=1141.820,254.150,-68.647,-177.525,8.026,148.832
C04570=1141.825,253.902,-68.620,-177.528,8.023,148.832
C04571=1141.828,253.653,-68.592,-177.531,8.020,148.832
C04572=1141.833,253.405,-68.563,-177.533,8.017,148.832
C04573=1141.838,253.156,-68.536,-177.536,8.014,148.832
C04574=1141.842,252.908,-68.508,-177.539,8.011,148.832
C04575=1141.846,252.660,-68.481,-177.542,8.008,148.832
C04576=1141.850,252.411,-68.453,-177.544,8.005,148.832
C04577=1141.855,252.163,-68.425,-177.547,8.002,148.833
C04578=1141.860,251.914,-68.398,-177.550,7.999,148.833
C04579=1141.864,251.666,-68.370,-177.553,7.997,148.833
C04580=1141.868,251.417,-68.342,-177.556,7.994,148.833
C04581=1141.872,251.168,-68.314,-177.558,7.991,148.833
C04582=1141.877,250.921,-68.287,-177.561,7.988,148.833
C04583=1141.881,250.672,-68.259,-177.564,7.985,148.833
C04584=1141.885,250.424,-68.231,-177.566,7.982,148.833
C04585=1141.890,250.175,-68.204,-177.569,7.979,148.833
C04586=1141.894,249.927,-68.176,-177.572,7.976,148.833
C04587=1141.899,249.679,-68.149,-177.575,7.973,148.833
C04588=1141.903,249.429,-68.122,-177.577,7.970,148.833
C04589=1141.907,249.182,-68.094,-177.580,7.967,148.833
C04590=1141.912,248.933,-68.067,-177.583,7.964,148.833
C04591=1141.915,248.685,-68.039,-177.586,7.961,148.833
C04592=1141.921,248.436,-68.011,-177.589,7.958,148.833
C04593=1141.925,248.187,-67.984,-177.591,7.955,148.833
C04594=1141.929,247.940,-67.957,-177.594,7.952,148.834
C04595=1141.933,247.690,-67.930,-177.597,7.949,148.834
C04596=1141.938,247.443,-67.902,-177.600,7.947,148.834
C04597=1141.942,247.194,-67.875,-177.603,7.944,148.834
C04598=1141.947,246.946,-67.848,-177.605,7.941,148.834
C04599=1141.951,246.696,-67.820,-177.608,7.938,148.834
C04600=1141.955,246.449,-67.793,-177.611,7.935,148.834
C04601=1141.960,246.200,-67.766,-177.614,7.932,148.834
C04602=1141.965,245.952,-67.738,-177.617,7.929,148.834
C04603=1141.969,245.702,-67.711,-177.619,7.926,148.834
C04604=1141.973,245.454,-67.683,-177.622,7.923,148.834
C04605=1141.978,245.206,-67.656,-177.624,7.920,148.834
C04606=1141.982,244.957,-67.629,-177.627,7.917,148.834
C04607=1141.987,244.709,-67.602,-177.630,7.914,148.834
C04608=1141.990,244.461,-67.575,-177.633,7.911,148.834
C04609=1141.995,244.212,-67.547,-177.636,7.908,148.834
C04610=1141.999,243.964,-67.520,-177.638,7.905,148.835
C04611=1142.004,243.715,-67.493,-177.641,7.902,148.835
C04612=1142.009,243.467,-67.466,-177.644,7.900,148.835
C04613=1142.013,243.218,-67.439,-177.647,7.897,148.835
C04614=1142.017,242.969,-67.412,-177.650,7.894,148.835
C04615=1142.021,242.721,-67.385,-177.652,7.891,148.835
C04616=1142.026,242.472,-67.358,-177.655,7.888,148.835
C04617=1142.031,242.224,-67.331,-177.658,7.885,148.835
C04618=1142.035,241.976,-67.303,-177.661,7.882,148.835
C04619=1142.039,241.728,-67.277,-177.664,7.879,148.835
C04620=1142.043,241.479,-67.250,-177.666,7.876,148.835
C04621=1142.047,241.230,-67.222,-177.669,7.873,148.835
C04622=1142.052,240.982,-67.195,-177.672,7.871,148.836
C04623=1142.056,240.733,-67.169,-177.675,7.868,148.836
C04624=1142.061,240.484,-67.143,-177.677,7.866,148.836
C04625=1142.066,240.236,-67.116,-177.680,7.863,148.836
C04626=1142.070,239.987,-67.088,-177.683,7.860,148.836
C04627=1142.074,239.739,-67.062,-177.686,7.857,148.836
C04628=1142.079,239.491,-67.035,-177.689,7.854,148.836
C04629=1142.084,239.242,-67.008,-177.691,7.851,148.836
C04630=1142.087,238.994,-66.981,-177.694,7.848,148.836
C04631=1142.092,238.745,-66.954,-177.697,7.845,148.836
C04632=1142.096,238.496,-66.927,-177.700,7.842,148.837
C04633=1142.100,238.247,-66.901,-177.703,7.839,148.837
C04634=1142.105,237.999,-66.874,-177.705,7.837,148.837
C04635=1142.110,237.750,-66.847,-177.708,7.834,148.837
C04636=1142.114,237.502,-66.821,-177.711,7.831,148.837
C04637=1142.118,237.254,-66.794,-177.714,7.828,148.837
C04638=1142.123,237.005,-66.768,-177.717,7.825,148.837
C04639=1142.127,236.756,-66.741,-177.719,7.822,148.837
C04640=1142.132,236.508,-66.714,-177.722,7.820,148.837
C04641=1142.136,236.260,-66.687,-177.724,7.817,148.837
C04642=1142.141,236.011,-66.661,-177.727,7.814,148.837
C04643=1142.145,235.739,-66.632,-177.731,7.811,148.838
C04644=1142.150,235.468,-66.603,-177.734,7.808,148.838
C04645=1142.155,235.195,-66.573,-177.737,7.805,148.838
C04646=1142.160,234.923,-66.544,-177.739,7.802,148.838
C04647=1142.164,234.675,-66.518,-177.742,7.799,148.838
C04648=1142.169,234.426,-66.492,-177.745,7.796,148.838
C04649=1142.173,234.178,-66.465,-177.748,7.793,148.838
C04650=1142.178,233.929,-66.438,-177.751,7.790,148.838
C04651=1142.182,233.680,-66.412,-177.754,7.788,148.838
C04652=1142.187,233.432,-66.385,-177.757,7.785,148.839
C04653=1142.191,233.183,-66.359,-177.759,7.782,148.839
C04654=1142.195,232.935,-66.333,-177.762,7.779,148.839
C04655=1142.200,232.686,-66.307,-177.765,7.776,148.839
C04656=1142.204,232.438,-66.280,-177.767,7.774,148.839
C04657=1142.209,232.190,-66.253,-177.770,7.771,148.839
C04658=1142.213,231.941,-66.228,-177.773,7.768,148.839
C04659=1142.218,231.693,-66.201,-177.776,7.765,148.839
C04660=1142.222,231.444,-66.175,-177.778,7.762,148.839
C04661=1142.226,231.195,-66.149,-177.782,7.760,148.840
C04662=1142.231,230.947,-66.122,-177.784,7.757,148.840
C04663=1142.235,230.698,-66.096,-177.787,7.754,148.840
C04664=1142.240,230.449,-66.069,-177.790,7.751,148.840
C04665=1142.244,230.200,-66.044,-177.792,7.749,148.840
C04666=1142.248,229.952,-66.017,-177.795,7.746,148.840
C04667=1142.253,229.704,-65.991,-177.798,7.743,148.840
C04668=1142.258,229.455,-65.965,-177.801,7.740,148.840
C04669=1142.262,229.207,-65.939,-177.804,7.737,148.841
C04670=1142.267,228.958,-65.913,-177.807,7.735,148.841
C04671=1142.271,228.709,-65.887,-177.810,7.732,148.841
C04672=1142.275,228.461,-65.860,-177.812,7.730,148.841
C04673=1142.280,228.212,-65.834,-177.815,7.727,148.841
C04674=1142.284,227.963,-65.809,-177.817,7.724,148.841
C04675=1142.289,227.715,-65.783,-177.820,7.721,148.841
C04676=1142.293,227.467,-65.756,-177.823,7.718,148.841
C04677=1142.298,227.217,-65.730,-177.826,7.715,148.841
C04678=1142.302,226.969,-65.704,-177.829,7.712,148.842
C04679=1142.307,226.720,-65.679,-177.831,7.710,148.842
C04680=1142.311,226.472,-65.652,-177.834,7.707,148.842
C04681=1142.315,226.223,-65.626,-177.837,7.704,148.842
C04682=1142.320,225.974,-65.600,-177.840,7.702,148.842
C04683=1142.324,225.726,-65.575,-177.843,7.699,148.842
C04684=1142.329,225.477,-65.549,-177.846,7.696,148.842
C04685=1142.333,225.229,-65.523,-177.849,7.693,148.842
C04686=1142.338,224.980,-65.496,-177.851,7.691,148.843
C04687=1142.342,224.731,-65.471,-177.854,7.688,148.843
C04688=1142.347,224.483,-65.445,-177.857,7.686,148.843
C04689=1142.351,224.234,-65.420,-177.860,7.683,148.843
C04690=1142.355,223.986,-65.394,-177.862,7.680,148.843
C04691=1142.359,223.737,-65.368,-177.865,7.677,148.843
C04692=1142.365,223.488,-65.342,-177.867,7.675,148.843
C04693=1142.369,223.240,-65.316,-177.870,7.672,148.843
C04694=1142.373,222.991,-65.291,-177.873,7.669,148.844
C04695=1142.378,222.742,-65.265,-177.876,7.666,148.844
C04696=1142.382,222.494,-65.239,-177.879,7.663,148.844
C04697=1142.387,222.245,-65.214,-177.882,7.661,148.844
C04698=1142.391,221.996,-65.188,-177.884,7.658,148.844
C04699=1142.396,221.748,-65.163,-177.887,7.656,148.844
C04700=1142.400,221.499,-65.137,-177.890,7.653,148.845
C04701=1142.404,221.251,-65.111,-177.893,7.650,148.845
C04702=1142.409,221.002,-65.086,-177.896,7.647,148.845
C04703=1142.413,220.754,-65.060,-177.898,7.645,148.845
C04704=1142.417,220.505,-65.034,-177.901,7.642,148.845
C04705=1142.423,220.256,-65.009,-177.904,7.640,148.845
C04706=1142.427,220.007,-64.984,-177.907,7.637,148.845
C04707=1142.431,219.759,-64.958,-177.910,7.634,148.845
C04708=1142.436,219.510,-64.933,-177.912,7.632,148.846
C04709=1142.440,219.262,-64.907,-177.915,7.629,148.846
C04710=1142.444,219.013,-64.881,-177.918,7.626,148.846
C04711=1142.449,218.764,-64.856,-177.921,7.623,148.846
C04712=1142.454,218.515,-64.831,-177.924,7.621,148.846
C04713=1142.458,218.266,-64.805,-177.926,7.619,148.847
C04714=1142.463,218.018,-64.779,-177.929,7.616,148.847
C04715=1142.467,217.769,-64.754,-177.932,7.613,148.847
C04716=1142.472,217.521,-64.729,-177.935,7.610,148.847
C04717=1142.476,217.272,-64.703,-177.938,7.607,148.847
C04718=1142.480,217.023,-64.678,-177.940,7.605,148.847
C04719=1142.486,216.775,-64.653,-177.943,7.602,148.847
C04720=1142.490,216.526,-64.627,-177.946,7.600,148.848
C04721=1142.494,216.278,-64.602,-177.949,7.597,148.848
C04722=1142.498,216.029,-64.577,-177.951,7.595,148.848
C04723=1142.503,215.780,-64.552,-177.954,7.592,148.848
C04724=1142.508,215.532,-64.526,-177.957,7.589,148.848
C04725=1142.512,215.282,-64.501,-177.960,7.586,148.848
C04726=1142.517,215.034,-64.476,-177.962,7.584,148.848
C04727=1142.521,214.785,-64.451,-177.965,7.581,148.849
C04728=1142.525,214.537,-64.426,-177.968,7.579,148.849
C04729=1142.530,214.288,-64.400,-177.971,7.576,148.849
C04730=1142.535,214.039,-64.376,-177.973,7.574,148.849
C04731=1142.539,213.791,-64.350,-177.977,7.571,148.849
C04732=1142.544,213.542,-64.325,-177.979,7.568,148.850
C04733=1142.548,213.293,-64.300,-177.982,7.565,148.850
C04734=1142.553,213.045,-64.275,-177.984,7.563,148.850
C04735=1142.557,212.796,-64.250,-177.988,7.561,148.850
C04736=1142.562,212.547,-64.225,-177.991,7.558,148.850
C04737=1142.566,212.299,-64.200,-177.993,7.555,148.850
C04738=1142.571,212.050,-64.175,-177.996,7.553,148.851
C04739=1142.575,211.800,-64.150,-177.999,7.550,148.851
C04740=1142.580,211.552,-64.125,-178.002,7.547,148.851
C04741=1142.584,211.303,-64.100,-178.004,7.544,148.851
C04742=1142.589,211.055,-64.075,-178.007,7.543,148.851
C04743=1142.593,210.806,-64.050,-178.010,7.540,148.851
C04744=1142.598,210.557,-64.026,-178.013,7.537,148.851
C04745=1142.602,210.308,-64.000,-178.016,7.534,148.852
C04746=1142.607,210.060,-63.975,-178.018,7.532,148.852
C04747=1142.612,209.789,-63.948,-178.021,7.530,148.852
C04748=1142.617,209.519,-63.921,-178.024,7.527,148.852
C04749=1142.621,209.248,-63.894,-178.027,7.524,148.852
C04750=1142.626,208.978,-63.868,-178.030,7.521,148.853
C04751=1142.631,208.728,-63.843,-178.033,7.518,148.853
C04752=1142.636,208.480,-63.817,-178.036,7.516,148.853
C04753=1142.640,208.231,-63.793,-178.039,7.513,148.853
C04754=1142.645,207.982,-63.768,-178.041,7.511,148.853
C04755=1142.649,207.734,-63.744,-178.045,7.508,148.854
C04756=1142.653,207.485,-63.718,-178.048,7.505,148.854
C04757=1142.658,207.237,-63.694,-178.050,7.503,148.854
C04758=1142.662,206.987,-63.669,-178.053,7.501,148.854
C04759=1142.667,206.738,-63.645,-178.056,7.498,148.854
C04760=1142.672,206.490,-63.620,-178.058,7.496,148.855
C04761=1142.676,206.241,-63.595,-178.061,7.493,148.855
C04762=1142.680,205.993,-63.571,-178.064,7.490,148.855
C04763=1142.686,205.744,-63.546,-178.067,7.487,148.855
C04764=1142.689,205.495,-63.522,-178.070,7.486,148.855
C04765=1142.694,205.246,-63.497,-178.072,7.483,148.856
C04766=1142.699,204.998,-63.473,-178.076,7.480,148.856
C04767=1142.703,204.748,-63.448,-178.078,7.478,148.856
C04768=1142.708,204.500,-63.424,-178.081,7.475,148.856
C04769=1142.713,204.251,-63.399,-178.084,7.473,148.856
C04770=1142.717,204.002,-63.375,-178.086,7.470,148.857
C04771=1142.722,203.753,-63.350,-178.089,7.468,148.857
C04772=1142.726,203.505,-63.326,-178.092,7.465,148.857
C04773=1142.731,203.256,-63.301,-178.094,7.463,148.857
C04774=1142.735,203.007,-63.277,-178.098,7.460,148.857
C04775=1142.740,202.759,-63.253,-178.101,7.457,148.858
C04776=1142.745,202.510,-63.228,-178.103,7.455,148.858
C04777=1142.749,202.261,-63.204,-178.106,7.453,148.858
C04778=1142.754,202.012,-63.179,-178.109,7.450,148.858
C04779=1142.758,201.764,-63.155,-178.112,7.448,148.858
C04780=1142.762,201.515,-63.131,-178.114,7.445,148.859
C04781=1142.767,201.266,-63.106,-178.118,7.443,148.859
C04782=1142.772,201.017,-63.082,-178.120,7.441,148.859
C04783=1142.776,200.769,-63.058,-178.123,7.438,148.859
C04784=1142.781,200.520,-63.034,-178.126,7.435,148.859
C04785=1142.785,200.271,-63.009,-178.128,7.433,148.860
C04786=1142.789,200.022,-62.985,-178.131,7.431,148.860
C04787=1142.794,199.774,-62.960,-178.134,7.428,148.860
C04788=1142.799,199.525,-62.937,-178.137,7.426,148.860
C04789=1142.803,199.275,-62.913,-178.140,7.423,148.860
C04790=1142.807,199.027,-62.889,-178.142,7.421,148.861
C04791=1142.813,198.778,-62.864,-178.145,7.418,148.861
C04792=1142.817,198.529,-62.840,-178.148,7.415,148.861
C04793=1142.822,198.281,-62.816,-178.151,7.414,148.861
C04794=1142.826,198.031,-62.791,-178.154,7.411,148.861
C04795=1142.831,197.783,-62.767,-178.157,7.408,148.862
C04796=1142.835,197.534,-62.744,-178.159,7.406,148.862
C04797=1142.840,197.286,-62.720,-178.162,7.403,148.862
C04798=1142.844,197.037,-62.696,-178.165,7.401,148.862
C04799=1142.849,196.788,-62.672,-178.167,7.399,148.863
C04800=1142.853,196.539,-62.647,-178.171,7.396,148.863
C04801=1142.858,196.290,-62.623,-178.173,7.394,148.863
C04802=1142.862,196.041,-62.600,-178.176,7.391,148.863
C04803=1142.867,195.793,-62.576,-178.178,7.389,148.863
C04804=1142.872,195.544,-62.552,-178.182,7.387,148.864
C04805=1142.877,195.295,-62.528,-178.184,7.384,148.864
C04806=1142.881,195.047,-62.504,-178.187,7.382,148.864
C04807=1142.885,194.797,-62.480,-178.190,7.379,148.864
C04808=1142.889,194.549,-62.456,-178.193,7.377,148.865
C04809=1142.894,194.300,-62.433,-178.195,7.375,148.865
C04810=1142.899,194.051,-62.408,-178.199,7.372,148.865
C04811=1142.904,193.802,-62.385,-178.201,7.370,148.865
C04812=1142.908,193.553,-62.361,-178.204,7.367,148.866
C04813=1142.913,193.304,-62.337,-178.206,7.365,148.866
C04814=1142.917,193.056,-62.313,-178.210,7.363,148.866
C04815=1142.922,192.807,-62.290,-178.213,7.360,148.866
C04816=1142.927,192.558,-62.266,-178.215,7.358,148.867
C04817=1142.931,192.309,-62.242,-178.218,7.355,148.867
C04818=1142.936,192.060,-62.219,-178.221,7.353,148.867
C04819=1142.940,191.812,-62.195,-178.224,7.351,148.867
C04820=1142.944,191.562,-62.171,-178.227,7.348,148.868
C04821=1142.949,191.314,-62.147,-178.229,7.346,148.868
C04822=1142.954,191.065,-62.124,-178.232,7.343,148.868
C04823=1142.958,190.816,-62.100,-178.235,7.341,148.868
C04824=1142.963,190.567,-62.076,-178.238,7.339,148.868
C04825=1142.967,190.318,-62.053,-178.240,7.337,148.869
C04826=1142.972,190.069,-62.030,-178.243,7.334,148.869
C04827=1142.976,189.821,-62.005,-178.246,7.331,148.869
C04828=1142.981,189.572,-61.982,-178.249,7.329,148.869
C04829=1142.986,189.323,-61.959,-178.252,7.327,148.870
C04830=1142.991,189.074,-61.935,-178.254,7.325,148.870
C04831=1142.995,188.825,-61.911,-178.257,7.322,148.870
C04832=1143.000,188.576,-61.888,-178.260,7.320,148.870
C04833=1143.004,188.327,-61.865,-178.263,7.317,148.870
C04834=1143.009,188.078,-61.841,-178.265,7.316,148.871
C04835=1143.013,187.830,-61.817,-178.268,7.313,148.871
C04836=1143.019,187.582,-61.794,-178.271,7.310,148.871
C04837=1143.023,187.333,-61.771,-178.274,7.308,148.872
C04838=1143.028,187.083,-61.747,-178.277,7.305,148.872
C04839=1143.033,186.834,-61.724,-178.280,7.304,148.872
C04840=1143.037,186.586,-61.701,-178.282,7.301,148.872
C04841=1143.041,186.337,-61.677,-178.285,7.299,148.873
C04842=1143.046,186.088,-61.654,-178.288,7.296,148.873
C04843=1143.051,185.839,-61.631,-178.291,7.294,148.873
C04844=1143.055,185.590,-61.607,-178.293,7.292,148.873
C04845=1143.060,185.341,-61.584,-178.296,7.290,148.874
C04846=1143.065,185.092,-61.560,-178.299,7.287,148.874
C04847=1143.069,184.843,-61.538,-178.302,7.285,148.874
C04848=1143.073,184.594,-61.514,-178.305,7.283,148.874
C04849=1143.078,184.345,-61.491,-178.307,7.281,148.875
C04850=1143.083,184.097,-61.468,-178.310,7.278,148.875
C04851=1143.087,183.827,-61.443,-178.314,7.275,148.875
C04852=1143.092,183.558,-61.417,-178.317,7.273,148.875
C04853=1143.098,183.288,-61.392,-178.319,7.271,148.876
C04854=1143.103,183.018,-61.367,-178.322,7.268,148.876
C04855=1143.107,182.769,-61.345,-178.325,7.265,148.876
C04856=1143.112,182.520,-61.321,-178.328,7.264,148.877
C04857=1143.116,182.271,-61.298,-178.331,7.261,148.877
C04858=1143.122,182.023,-61.275,-178.334,7.259,148.877
C04859=1143.126,181.774,-61.252,-178.337,7.257,148.877
C04860=1143.130,181.525,-61.229,-178.339,7.254,148.877
C04861=1143.135,181.276,-61.206,-178.342,7.252,148.878
C04862=1143.139,181.027,-61.183,-178.345,7.250,148.878
C04863=1143.144,180.778,-61.160,-178.348,7.247,148.878
C04864=1143.149,180.530,-61.137,-178.351,7.246,148.879
C04865=1143.153,180.281,-61.114,-178.353,7.243,148.879
C04866=1143.158,180.032,-61.091,-178.356,7.241,148.879
C04867=1143.163,179.783,-61.068,-178.359,7.238,148.880
C04868=1143.167,179.533,-61.046,-178.362,7.236,148.880
C04869=1143.172,179.285,-61.023,-178.365,7.234,148.880
C04870=1143.177,179.036,-60.999,-178.367,7.232,148.880
C04871=1143.181,178.787,-60.976,-178.370,7.230,148.881
C04872=1143.186,178.538,-60.954,-178.373,7.227,148.881
C04873=1143.190,178.289,-60.931,-178.375,7.225,148.881
C04874=1143.195,178.041,-60.908,-178.379,7.223,148.881
C04875=1143.200,177.792,-60.885,-178.381,7.221,148.882
C04876=1143.204,177.542,-60.863,-178.384,7.218,148.882
C04877=1143.209,177.293,-60.839,-178.387,7.216,148.882
C04878=1143.213,177.045,-60.817,-178.390,7.214,148.883
C04879=1143.218,176.796,-60.794,-178.392,7.212,148.883
C04880=1143.222,176.547,-60.771,-178.396,7.209,148.883
C04881=1143.227,176.297,-60.749,-178.398,7.207,148.883
C04882=1143.232,176.049,-60.726,-178.401,7.205,148.884
C04883=1143.237,175.800,-60.703,-178.404,7.203,148.884
C04884=1143.241,175.551,-60.681,-178.406,7.201,148.884
C04885=1143.246,175.302,-60.658,-178.409,7.198,148.884
C04886=1143.250,175.053,-60.636,-178.412,7.197,148.885
C04887=1143.255,174.804,-60.613,-178.415,7.194,148.885
C04888=1143.260,174.556,-60.590,-178.417,7.192,148.885
C04889=1143.265,174.306,-60.568,-178.421,7.189,148.886
C04890=1143.269,174.058,-60.545,-178.423,7.187,148.886
C04891=1143.274,173.808,-60.522,-178.426,7.185,148.886
C04892=1143.278,173.560,-60.500,-178.429,7.183,148.886
C04893=1143.283,173.310,-60.477,-178.431,7.181,148.887
C04894=1143.287,173.062,-60.454,-178.435,7.178,148.887
C04895=1143.292,172.813,-60.433,-178.437,7.177,148.887
C04896=1143.297,172.563,-60.410,-178.440,7.174,148.887
C04897=1143.302,172.315,-60.388,-178.443,7.172,148.888
C04898=1143.307,172.066,-60.365,-178.446,7.170,148.888
C04899=1143.311,171.817,-60.342,-178.449,7.168,148.889
C04900=1143.315,171.568,-60.320,-178.451,7.166,148.889
C04901=1143.320,171.319,-60.297,-178.454,7.163,148.889
C04902=1143.324,171.070,-60.275,-178.457,7.161,148.889
C04903=1143.329,170.821,-60.253,-178.460,7.159,148.890
C04904=1143.334,170.572,-60.230,-178.462,7.157,148.890
C04905=1143.339,170.324,-60.208,-178.465,7.155,148.890
C04906=1143.343,170.074,-60.186,-178.468,7.152,148.890
C04907=1143.348,169.825,-60.163,-178.471,7.150,148.891
C04908=1143.353,169.577,-60.141,-178.474,7.148,148.891
C04909=1143.357,169.327,-60.119,-178.477,7.146,148.892
C04910=1143.363,169.078,-60.097,-178.479,7.144,148.892
C04911=1143.367,168.830,-60.074,-178.482,7.142,148.892
C04912=1143.371,168.581,-60.053,-178.485,7.140,148.892
C04913=1143.376,168.331,-60.030,-178.488,7.137,148.893
C04914=1143.381,168.082,-60.008,-178.490,7.135,148.893
C04915=1143.385,167.834,-59.985,-178.493,7.134,148.893
C04916=1143.390,167.585,-59.963,-178.496,7.131,148.894
C04917=1143.395,167.336,-59.941,-178.499,7.129,148.894
C04918=1143.399,167.086,-59.919,-178.502,7.126,148.894
C04919=1143.404,166.838,-59.897,-178.505,7.125,148.895
C04920=1143.408,166.589,-59.875,-178.507,7.123,148.895
C04921=1143.414,166.340,-59.852,-178.510,7.120,148.895
C04922=1143.418,166.091,-59.830,-178.513,7.118,148.895
C04923=1143.423,165.842,-59.809,-178.516,7.117,148.896
C04924=1143.427,165.593,-59.787,-178.518,7.114,148.896
C04925=1143.432,165.344,-59.765,-178.521,7.112,148.896
C04926=1143.436,165.095,-59.743,-178.524,7.109,148.897
C04927=1143.442,164.846,-59.721,-178.527,7.108,148.897
C04928=1143.446,164.596,-59.698,-178.529,7.106,148.897
C04929=1143.451,164.348,-59.677,-178.533,7.103,148.898
C04930=1143.455,164.098,-59.655,-178.535,7.101,148.898
C04931=1143.460,163.850,-59.632,-178.538,7.100,148.898
C04932=1143.464,163.601,-59.610,-178.541,7.097,148.898
C04933=1143.469,163.352,-59.589,-178.544,7.095,148.899
C04934=1143.473,163.103,-59.567,-178.546,7.093,148.899
C04935=1143.478,162.854,-59.545,-178.550,7.091,148.900
C04936=1143.484,162.604,-59.523,-178.552,7.089,148.900
C04937=1143.488,162.356,-59.501,-178.554,7.087,148.900
C04938=1143.493,162.107,-59.480,-178.558,7.084,148.900
C04939=1143.498,161.858,-59.458,-178.560,7.083,148.901
C04940=1143.502,161.609,-59.436,-178.563,7.081,148.901
C04941=1143.507,161.360,-59.414,-178.566,7.078,148.901
C04942=1143.512,161.111,-59.392,-178.569,7.076,148.902
C04943=1143.516,160.862,-59.370,-178.571,7.075,148.902
C04944=1143.521,160.613,-59.348,-178.575,7.072,148.902
C04945=1143.526,160.364,-59.327,-178.577,7.070,148.903
C04946=1143.530,160.114,-59.305,-178.580,7.068,148.903
C04947=1143.535,159.866,-59.284,-178.583,7.066,148.903
C04948=1143.540,159.617,-59.262,-178.586,7.064,148.904
C04949=1143.544,159.368,-59.240,-178.588,7.062,148.904
C04950=1143.549,159.119,-59.218,-178.591,7.060,148.904
C04951=1143.553,158.870,-59.196,-178.594,7.058,148.905
C04952=1143.558,158.621,-59.175,-178.597,7.056,148.905
C04953=1143.563,158.372,-59.154,-178.600,7.054,148.905
C04954=1143.568,158.123,-59.132,-178.602,7.051,148.905
C04955=1143.572,157.853,-59.109,-178.605,7.049,148.906
C04956=1143.578,157.584,-59.085,-178.608,7.047,148.906
C04957=1143.583,157.316,-59.062,-178.611,7.045,148.907
C04958=1143.588,157.047,-59.039,-178.614,7.043,148.907
C04959=1143.593,156.798,-59.017,-178.617,7.040,148.907
C04960=1143.598,156.548,-58.996,-178.620,7.039,148.908
C04961=1143.602,156.300,-58.975,-178.623,7.037,148.908
C04962=1143.606,156.051,-58.953,-178.626,7.035,148.908
C04963=1143.611,155.802,-58.932,-178.628,7.032,148.909
C04964=1143.616,155.553,-58.910,-178.631,7.031,148.909
C04965=1143.621,155.304,-58.888,-178.634,7.029,148.909
C04966=1143.626,155.054,-58.867,-178.637,7.026,148.910
C04967=1143.631,154.806,-58.845,-178.640,7.025,148.910
C04968=1143.635,154.557,-58.825,-178.642,7.023,148.910
C04969=1143.639,154.307,-58.803,-178.645,7.021,148.911
C04970=1143.644,154.059,-58.781,-178.648,7.018,148.911
C04971=1143.649,153.809,-58.760,-178.651,7.017,148.911
C04972=1143.654,153.561,-58.739,-178.653,7.015,148.912
C04973=1143.658,153.311,-58.718,-178.657,7.012,148.912
C04974=1143.663,153.063,-58.696,-178.659,7.010,148.912
C04975=1143.668,152.813,-58.675,-178.662,7.009,148.913
C04976=1143.673,152.565,-58.654,-178.664,7.007,148.913
C04977=1143.678,152.315,-58.632,-178.668,7.004,148.913
C04978=1143.682,152.066,-58.611,-178.670,7.003,148.914
C04979=1143.687,151.817,-58.590,-178.673,7.001,148.914
C04980=1143.692,151.568,-58.569,-178.676,6.999,148.915
C04981=1143.696,151.319,-58.548,-178.679,6.996,148.915
C04982=1143.701,151.070,-58.527,-178.681,6.995,148.915
C04983=1143.706,150.821,-58.505,-178.684,6.993,148.915
C04984=1143.711,150.572,-58.484,-178.687,6.991,148.916
C04985=1143.715,150.323,-58.464,-178.690,6.989,148.916
C04986=1143.720,150.074,-58.442,-178.693,6.987,148.917
C04987=1143.725,149.824,-58.421,-178.695,6.985,148.917
C04988=1143.729,149.576,-58.400,-178.698,6.983,148.917
C04989=1143.734,149.326,-58.379,-178.701,6.981,148.918
C04990=1143.739,149.077,-58.358,-178.704,6.979,148.918
C04991=1143.744,148.828,-58.337,-178.706,6.977,148.918
C04992=1143.748,148.580,-58.316,-178.709,6.976,148.919
C04993=1143.753,148.330,-58.294,-178.712,6.973,148.919
C04994=1143.757,148.081,-58.274,-178.715,6.971,148.919
C04995=1143.762,147.832,-58.252,-178.718,6.970,148.920
C04996=1143.767,147.583,-58.232,-178.720,6.968,148.920
C04997=1143.772,147.334,-58.211,-178.723,6.965,148.920
C04998=1143.777,147.085,-58.190,-178.726,6.963,148.921
C04999=1143.781,146.836,-58.169,-178.729,6.962,148.921
C05000=1143.786,146.587,-58.148,-178.732,6.960,148.922
C05001=1143.790,146.337,-58.127,-178.734,6.958,148.922
C05002=1143.795,146.088,-58.106,-178.738,6.956,148.922
C05003=1143.800,145.839,-58.086,-178.740,6.954,148.923
C05004=1143.805,145.590,-58.065,-178.743,6.952,148.923
C05005=1143.810,145.341,-58.043,-178.745,6.950,148.923
C05006=1143.814,145.092,-58.023,-178.749,6.948,148.924
C05007=1143.819,144.843,-58.002,-178.751,6.946,148.924
C05008=1143.824,144.594,-57.982,-178.754,6.944,148.924
C05009=1143.829,144.345,-57.961,-178.757,6.943,148.925
C05010=1143.834,144.096,-57.940,-178.759,6.941,148.925
C05011=1143.839,143.847,-57.919,-178.763,6.938,148.925
C05012=1143.843,143.598,-57.899,-178.765,6.937,148.926
C05013=1143.847,143.348,-57.878,-178.768,6.935,148.926
C05014=1143.852,143.099,-57.857,-178.771,6.933,148.927
C05015=1143.857,142.850,-57.837,-178.773,6.931,148.927
C05016=1143.862,142.601,-57.816,-178.776,6.929,148.927
C05017=1143.866,142.352,-57.795,-178.779,6.927,148.928
C05018=1143.871,142.102,-57.775,-178.782,6.925,148.928
C05019=1143.876,141.853,-57.754,-178.784,6.923,148.928
C05020=1143.881,141.604,-57.733,-178.787,6.922,148.929
C05021=1143.885,141.355,-57.713,-178.790,6.920,148.929
C05022=1143.890,141.106,-57.692,-178.793,6.918,148.930
C05023=1143.895,140.857,-57.671,-178.796,6.916,148.930
C05024=1143.899,140.608,-57.651,-178.799,6.914,148.930
C05025=1143.904,140.359,-57.631,-178.801,6.912,148.931
C05026=1143.909,140.110,-57.610,-178.804,6.911,148.931
C05027=1143.914,139.861,-57.589,-178.807,6.909,148.931
C05028=1143.919,139.612,-57.568,-178.810,6.906,148.932
C05029=1143.923,139.363,-57.548,-178.812,6.904,148.932
C05030=1143.928,139.114,-57.528,-178.815,6.903,148.932
C05031=1143.933,138.864,-57.507,-178.818,6.901,148.933
C05032=1143.937,138.615,-57.487,-178.820,6.899,148.933
C05033=1143.942,138.366,-57.467,-178.823,6.898,148.934
C05034=1143.947,138.118,-57.447,-178.827,6.895,148.934
C05035=1143.952,137.868,-57.426,-178.829,6.893,148.934
C05036=1143.957,137.619,-57.406,-178.832,6.892,148.935
C05037=1143.961,137.370,-57.386,-178.835,6.890,148.935
C05038=1143.966,137.121,-57.365,-178.837,6.888,148.936
C05039=1143.971,136.872,-57.344,-178.840,6.887,148.936
C05040=1143.976,136.622,-57.325,-178.843,6.885,148.936
C05041=1143.980,136.373,-57.304,-178.846,6.882,148.937
C05042=1143.985,136.124,-57.283,-178.849,6.881,148.937
C05043=1143.990,135.875,-57.263,-178.852,6.879,148.937
C05044=1143.994,135.625,-57.243,-178.854,6.877,148.938
C05045=1143.999,135.376,-57.223,-178.857,6.875,148.938
C05046=1144.005,135.128,-57.202,-178.860,6.874,148.939
C05047=1144.009,134.878,-57.183,-178.862,6.872,148.939
C05048=1144.014,134.629,-57.162,-178.866,6.870,148.939
C05049=1144.018,134.380,-57.142,-178.868,6.868,148.940
C05050=1144.023,134.131,-57.122,-178.871,6.866,148.940
C05051=1144.027,133.882,-57.102,-178.874,6.864,148.941
C05052=1144.033,133.633,-57.081,-178.876,6.862,148.941
C05053=1144.038,133.384,-57.062,-178.879,6.861,148.941
C05054=1144.042,133.135,-57.041,-178.882,6.859,148.942
C05055=1144.047,132.885,-57.022,-178.884,6.857,148.942
C05056=1144.052,132.636,-57.001,-178.888,6.855,148.942
C05057=1144.056,132.387,-56.982,-178.890,6.853,148.943
C05058=1144.062,132.138,-56.961,-178.893,6.851,148.943
C05059=1144.066,131.869,-56.940,-178.896,6.850,148.944
C05060=1144.071,131.601,-56.918,-178.899,6.848,148.944
C05061=1144.077,131.332,-56.896,-178.902,6.846,148.945
C05062=1144.082,131.064,-56.875,-178.905,6.844,148.945
C05063=1144.087,130.815,-56.855,-178.908,6.842,148.945
C05064=1144.091,130.565,-56.835,-178.910,6.841,148.946
C05065=1144.096,130.316,-56.815,-178.913,6.839,148.946
C05066=1144.101,130.067,-56.795,-178.916,6.836,148.946
C05067=1144.107,129.818,-56.775,-178.919,6.835,148.947
C05068=1144.111,129.569,-56.755,-178.922,6.833,148.947
C05069=1144.116,129.319,-56.735,-178.925,6.831,148.948
C05070=1144.120,129.070,-56.715,-178.927,6.830,148.948
C05071=1144.126,128.821,-56.696,-178.930,6.828,148.948
C05072=1144.130,128.572,-56.676,-178.933,6.826,148.949
C05073=1144.135,128.323,-56.656,-178.935,6.825,148.949
C05074=1144.140,128.073,-56.636,-178.938,6.823,148.950
C05075=1144.145,127.825,-56.616,-178.941,6.821,148.950
C05076=1144.149,127.575,-56.596,-178.944,6.819,148.950
C05077=1144.154,127.326,-56.577,-178.946,6.818,148.951
C05078=1144.159,127.076,-56.557,-178.949,6.816,148.951
C05079=1144.164,126.828,-56.537,-178.952,6.814,148.952
C05080=1144.169,126.579,-56.517,-178.955,6.812,148.952
C05081=1144.173,126.329,-56.498,-178.958,6.810,148.952
C05082=1144.178,126.081,-56.478,-178.961,6.808,148.953
C05083=1144.182,125.831,-56.459,-178.963,6.807,148.953
C05084=1144.187,125.582,-56.439,-178.966,6.805,148.954
C05085=1144.192,125.332,-56.419,-178.969,6.803,148.954
C05086=1144.197,125.084,-56.399,-178.971,6.802,148.954
C05087=1144.202,124.834,-56.380,-178.974,6.800,148.955
C05088=1144.206,124.585,-56.360,-178.977,6.798,148.955
C05089=1144.212,124.336,-56.341,-178.980,6.797,148.956
C05090=1144.216,124.086,-56.321,-178.982,6.795,148.956
C05091=1144.220,123.837,-56.302,-178.986,6.794,148.957
C05092=1144.226,123.589,-56.282,-178.988,6.792,148.957
C05093=1144.230,123.339,-56.262,-178.991,6.790,148.957
C05094=1144.235,123.090,-56.243,-178.994,6.788,148.958
C05095=1144.240,122.841,-56.223,-178.996,6.787,148.958
C05096=1144.245,122.591,-56.204,-178.999,6.785,148.959
C05097=1144.249,122.342,-56.185,-179.002,6.783,148.959
C05098=1144.254,122.093,-56.165,-179.005,6.782,148.959
C05099=1144.259,121.844,-56.146,-179.007,6.780,148.960
C05100=1144.265,121.595,-56.126,-179.011,6.777,148.960
C05101=1144.269,121.346,-56.106,-179.013,6.776,148.961
C05102=1144.273,121.097,-56.087,-179.016,6.774,148.961
C05103=1144.278,120.848,-56.068,-179.019,6.772,148.961
C05104=1144.283,120.598,-56.048,-179.022,6.771,148.962
C05105=1144.288,120.349,-56.029,-179.024,6.769,148.962
C05106=1144.292,120.100,-56.010,-179.027,6.767,148.963
C05107=1144.297,119.851,-55.990,-179.030,6.766,148.963
C05108=1144.302,119.602,-55.971,-179.032,6.764,148.963
C05109=1144.307,119.352,-55.951,-179.036,6.763,148.964
C05110=1144.312,119.103,-55.933,-179.038,6.761,148.964
C05111=1144.317,118.853,-55.913,-179.041,6.759,148.965
C05112=1144.322,118.604,-55.894,-179.044,6.758,148.965
C05113=1144.327,118.355,-55.875,-179.046,6.756,148.966
C05114=1144.332,118.106,-55.856,-179.049,6.754,148.966
C05115=1144.336,117.857,-55.836,-179.052,6.752,148.966
C05116=1144.341,117.607,-55.817,-179.055,6.751,148.967
C05117=1144.346,117.359,-55.798,-179.057,6.749,148.967
C05118=1144.350,117.109,-55.778,-179.060,6.747,148.968
C05119=1144.356,116.860,-55.759,-179.063,6.746,148.968
C05120=1144.360,116.610,-55.741,-179.066,6.744,148.969
C05121=1144.365,116.361,-55.721,-179.068,6.742,148.969
C05122=1144.370,116.112,-55.702,-179.072,6.741,148.970
C05123=1144.375,115.863,-55.683,-179.074,6.739,148.970
C05124=1144.380,115.614,-55.663,-179.077,6.738,148.970
C05125=1144.384,115.365,-55.645,-179.080,6.736,148.971
C05126=1144.389,115.115,-55.626,-179.082,6.734,148.971
C05127=1144.395,114.866,-55.606,-179.085,6.732,148.972
C05128=1144.399,114.617,-55.587,-179.087,6.732,148.972
C05129=1144.404,114.367,-55.569,-179.090,6.730,148.972
C05130=1144.408,114.118,-55.550,-179.093,6.728,148.973
C05131=1144.414,113.869,-55.530,-179.095,6.727,148.973
C05132=1144.418,113.621,-55.512,-179.099,6.725,148.974
C05133=1144.423,113.371,-55.493,-179.101,6.724,148.974
C05134=1144.429,113.122,-55.473,-179.104,6.722,148.975
C05135=1144.433,112.872,-55.454,-179.107,6.720,148.975
C05136=1144.438,112.623,-55.436,-179.110,6.718,148.975
C05137=1144.442,112.374,-55.417,-179.112,6.717,148.976
C05138=1144.448,112.125,-55.397,-179.115,6.715,148.976
C05139=1144.452,111.876,-55.379,-179.118,6.713,148.977
C05140=1144.457,111.626,-55.360,-179.120,6.712,148.977
C05141=1144.462,111.377,-55.342,-179.123,6.710,148.977
C05142=1144.467,111.127,-55.322,-179.126,6.709,148.978
C05143=1144.471,110.879,-55.303,-179.129,6.707,148.979
C05144=1144.477,110.629,-55.285,-179.132,6.705,148.979
C05145=1144.481,110.380,-55.266,-179.135,6.704,148.979
C05146=1144.487,110.131,-55.247,-179.137,6.702,148.980
C05147=1144.491,109.881,-55.228,-179.140,6.700,148.980
C05148=1144.496,109.632,-55.210,-179.143,6.699,148.981
C05149=1144.501,109.383,-55.191,-179.146,6.697,148.981
C05150=1144.505,109.133,-55.173,-179.148,6.696,148.982
C05151=1144.511,108.885,-55.153,-179.151,6.695,148.982
C05152=1144.515,108.635,-55.135,-179.154,6.693,148.982
C05153=1144.520,108.386,-55.116,-179.156,6.691,148.983
C05154=1144.525,108.137,-55.098,-179.159,6.690,148.983
C05155=1144.529,107.887,-55.079,-179.162,6.688,148.984
C05156=1144.535,107.638,-55.060,-179.164,6.686,148.984
C05157=1144.539,107.389,-55.041,-179.168,6.685,148.985
C05158=1144.544,107.139,-55.023,-179.170,6.683,148.985
C05159=1144.549,106.891,-55.004,-179.173,6.682,148.986
C05160=1144.554,106.641,-54.986,-179.176,6.680,148.986
C05161=1144.558,106.391,-54.967,-179.179,6.678,148.986
C05162=1144.564,106.143,-54.948,-179.181,6.677,148.987
C05163=1144.569,105.874,-54.929,-179.185,6.675,148.987
C05164=1144.575,105.606,-54.909,-179.187,6.673,148.988
C05165=1144.579,105.337,-54.888,-179.190,6.672,148.988
C05166=1144.585,105.069,-54.868,-179.193,6.670,148.989
C05167=1144.590,104.820,-54.850,-179.196,6.669,148.989
C05168=1144.594,104.571,-54.832,-179.199,6.667,148.990
C05169=1144.599,104.321,-54.813,-179.201,6.665,148.990
C05170=1144.604,104.072,-54.795,-179.204,6.664,148.991
C05171=1144.609,103.823,-54.777,-179.206,6.663,148.991
C05172=1144.614,103.574,-54.758,-179.209,6.661,148.991
C05173=1144.619,103.324,-54.739,-179.212,6.660,148.992
C05174=1144.624,103.075,-54.721,-179.215,6.658,148.992
C05175=1144.628,102.826,-54.703,-179.218,6.656,148.993
C05176=1144.633,102.577,-54.684,-179.220,6.655,148.993
C05177=1144.637,102.327,-54.666,-179.223,6.653,148.994
C05178=1144.643,102.078,-54.647,-179.226,6.651,148.994
C05179=1144.648,101.828,-54.629,-179.229,6.650,148.995
C05180=1144.653,101.579,-54.611,-179.231,6.649,148.995
C05181=1144.657,101.330,-54.592,-179.234,6.648,148.996
C05182=1144.663,101.081,-54.574,-179.237,6.646,148.996
C05183=1144.667,100.831,-54.556,-179.239,6.644,148.996
C05184=1144.672,100.582,-54.538,-179.242,6.642,148.997
C05185=1144.677,100.333,-54.520,-179.245,6.641,148.997
C05186=1144.682,100.083,-54.501,-179.248,6.639,148.998
C05187=1144.686,99.834,-54.484,-179.250,6.639,148.998
C05188=1144.691,99.585,-54.466,-179.253,6.637,148.999
C05189=1144.697,99.336,-54.446,-179.256,6.635,148.999
C05190=1144.702,99.087,-54.428,-179.258,6.634,148.999
C05191=1144.707,98.838,-54.410,-179.262,6.632,149.000
C05192=1144.711,98.588,-54.392,-179.264,6.631,149.001
C05193=1144.716,98.338,-54.374,-179.267,6.629,149.001
C05194=1144.721,98.089,-54.356,-179.269,6.628,149.001
C05195=1144.726,97.840,-54.338,-179.272,6.626,149.002
C05196=1144.731,97.591,-54.320,-179.275,6.625,149.002
C05197=1144.735,97.342,-54.302,-179.278,6.623,149.003
C05198=1144.740,97.092,-54.284,-179.281,6.622,149.003
C05199=1144.745,96.843,-54.266,-179.283,6.620,149.004
C05200=1144.750,96.593,-54.247,-179.286,6.618,149.004
C05201=1144.755,96.344,-54.229,-179.289,6.618,149.005
C05202=1144.760,96.095,-54.211,-179.292,6.616,149.005
C05203=1144.765,95.846,-54.193,-179.294,6.614,149.006
C05204=1144.770,95.597,-54.175,-179.297,6.613,149.006
C05205=1144.775,95.347,-54.157,-179.300,6.611,149.006
C05206=1144.779,95.097,-54.140,-179.302,6.609,149.007
C05207=1144.784,94.848,-54.122,-179.305,6.609,149.007
C05208=1144.789,94.599,-54.104,-179.308,6.607,149.008
C05209=1144.794,94.349,-54.086,-179.311,6.606,149.008
C05210=1144.799,94.100,-54.068,-179.313,6.604,149.009
C05211=1144.804,93.851,-54.050,-179.316,6.603,149.009
C05212=1144.809,93.602,-54.032,-179.319,6.602,149.010
C05213=1144.814,93.352,-54.014,-179.321,6.600,149.010
C05214=1144.819,93.103,-53.996,-179.324,6.598,149.011
C05215=1144.823,92.854,-53.979,-179.327,6.597,149.011
C05216=1144.828,92.605,-53.961,-179.330,6.595,149.012
C05217=1144.833,92.356,-53.943,-179.332,6.594,149.012
C05218=1144.838,92.106,-53.925,-179.335,6.593,149.013
C05219=1144.843,91.857,-53.908,-179.338,6.591,149.013
C05220=1144.848,91.607,-53.890,-179.340,6.589,149.013
C05221=1144.853,91.358,-53.872,-179.344,6.588,149.014
C05222=1144.857,91.108,-53.854,-179.346,6.587,149.014
C05223=1144.863,90.859,-53.836,-179.348,6.586,149.015
C05224=1144.867,90.609,-53.818,-179.351,6.584,149.015
C05225=1144.872,90.360,-53.800,-179.354,6.583,149.016
C05226=1144.877,90.111,-53.784,-179.357,6.581,149.016
C05227=1144.882,89.862,-53.766,-179.359,6.580,149.017
C05228=1144.887,89.612,-53.748,-179.362,6.578,149.017
C05229=1144.892,89.363,-53.730,-179.365,6.577,149.018
C05230=1144.897,89.113,-53.713,-179.368,6.575,149.018
C05231=1144.902,88.864,-53.695,-179.371,6.574,149.019
C05232=1144.906,88.615,-53.678,-179.373,6.573,149.019
C05233=1144.911,88.366,-53.660,-179.376,6.571,149.020
C05234=1144.917,88.117,-53.642,-179.379,6.570,149.020
C05235=1144.922,87.867,-53.625,-179.382,6.568,149.021
C05236=1144.927,87.618,-53.607,-179.384,6.567,149.021
C05237=1144.931,87.369,-53.590,-179.386,6.566,149.021
C05238=1144.936,87.120,-53.572,-179.390,6.564,149.022
C05239=1144.941,86.870,-53.554,-179.392,6.563,149.023
C05240=1144.946,86.621,-53.537,-179.395,6.561,149.023
C05241=1144.950,86.372,-53.520,-179.397,6.560,149.023
C05242=1144.956,86.122,-53.502,-179.400,6.559,149.024
C05243=1144.961,85.873,-53.484,-179.403,6.557,149.024
C05244=1144.966,85.623,-53.467,-179.406,6.556,149.025
C05245=1144.970,85.374,-53.450,-179.408,6.555,149.025
C05246=1144.975,85.124,-53.433,-179.411,6.553,149.026
C05247=1144.980,84.875,-53.415,-179.414,6.552,149.026
C05248=1144.985,84.625,-53.397,-179.417,6.550,149.027
C05249=1144.990,84.377,-53.380,-179.419,6.549,149.027
C05250=1144.995,84.127,-53.363,-179.422,6.547,149.028
C05251=1145.001,83.878,-53.346,-179.425,6.546,149.028
C05252=1145.005,83.629,-53.328,-179.428,6.545,149.029
C05253=1145.010,83.379,-53.311,-179.430,6.544,149.029
C05254=1145.015,83.130,-53.293,-179.433,6.542,149.030
C05255=1145.019,82.880,-53.276,-179.436,6.541,149.030
C05256=1145.024,82.631,-53.259,-179.438,6.540,149.031
C05257=1145.029,82.381,-53.241,-179.441,6.538,149.031
C05258=1145.035,82.132,-53.225,-179.443,6.536,149.031
C05259=1145.039,81.883,-53.207,-179.447,6.535,149.032
C05260=1145.044,81.634,-53.190,-179.449,6.534,149.033
C05261=1145.049,81.384,-53.173,-179.452,6.533,149.033
C05262=1145.054,81.135,-53.155,-179.455,6.531,149.034
C05263=1145.059,80.885,-53.138,-179.458,6.530,149.034
C05264=1145.064,80.636,-53.121,-179.460,6.529,149.035
C05265=1145.069,80.387,-53.104,-179.462,6.527,149.035
C05266=1145.074,80.138,-53.087,-179.466,6.526,149.036
C05267=1145.079,79.869,-53.068,-179.468,6.524,149.036
C05268=1145.084,79.601,-53.050,-179.471,6.523,149.036
C05269=1145.090,79.332,-53.032,-179.474,6.522,149.037
C05270=1145.095,79.063,-53.013,-179.476,6.520,149.038
C05271=1145.100,78.815,-52.996,-179.480,6.519,149.038
C05272=1145.105,78.565,-52.979,-179.482,6.517,149.039
C05273=1145.110,78.316,-52.962,-179.485,6.516,149.039
C05274=1145.115,78.066,-52.945,-179.487,6.515,149.039
C05275=1145.120,77.817,-52.928,-179.491,6.514,149.040
C05276=1145.125,77.568,-52.911,-179.493,6.512,149.041
C05277=1145.129,77.318,-52.894,-179.495,6.511,149.041
C05278=1145.135,77.069,-52.877,-179.499,6.510,149.042
C05279=1145.140,76.820,-52.860,-179.501,6.508,149.042
C05280=1145.145,76.570,-52.843,-179.504,6.507,149.042
C05281=1145.149,76.321,-52.826,-179.506,6.506,149.043
C05282=1145.155,76.071,-52.809,-179.510,6.504,149.044
C05283=1145.159,75.823,-52.792,-179.512,6.503,149.044
C05284=1145.165,75.573,-52.775,-179.514,6.502,149.044
C05285=1145.169,75.323,-52.758,-179.518,6.500,149.045
C05286=1145.173,75.074,-52.741,-179.520,6.500,149.046
C05287=1145.179,74.825,-52.725,-179.523,6.498,149.046
C05288=1145.184,74.575,-52.708,-179.525,6.496,149.046
C05289=1145.189,74.326,-52.691,-179.529,6.495,149.047
C05290=1145.193,74.076,-52.674,-179.531,6.494,149.047
C05291=1145.199,73.827,-52.658,-179.533,6.492,149.048
C05292=1145.204,73.577,-52.640,-179.537,6.491,149.049
C05293=1145.208,73.328,-52.624,-179.539,6.490,149.049
C05294=1145.214,73.079,-52.607,-179.542,6.489,149.049
C05295=1145.219,72.829,-52.590,-179.544,6.487,149.050
C05296=1145.223,72.580,-52.573,-179.547,6.486,149.050
C05297=1145.229,72.331,-52.557,-179.550,6.485,149.051
C05298=1145.233,72.081,-52.540,-179.552,6.483,149.051
C05299=1145.238,71.832,-52.523,-179.555,6.483,149.052
C05300=1145.244,71.583,-52.506,-179.558,6.481,149.052
C05301=1145.248,71.333,-52.490,-179.560,6.480,149.053
C05302=1145.253,71.084,-52.473,-179.563,6.479,149.054
C05303=1145.258,70.835,-52.456,-179.566,6.477,149.054
C05304=1145.263,70.585,-52.440,-179.568,6.476,149.054
C05305=1145.268,70.335,-52.423,-179.571,6.475,149.055
C05306=1145.274,70.086,-52.407,-179.574,6.473,149.055
C05307=1145.278,69.837,-52.390,-179.576,6.473,149.056
C05308=1145.282,69.587,-52.373,-179.579,6.471,149.056
C05309=1145.288,69.338,-52.356,-179.582,6.470,149.057
C05310=1145.293,69.088,-52.340,-179.584,6.469,149.057
C05311=1145.298,68.839,-52.324,-179.587,6.467,149.058
C05312=1145.303,68.590,-52.307,-179.590,6.466,149.059
C05313=1145.308,68.340,-52.290,-179.592,6.465,149.059
C05314=1145.313,68.091,-52.274,-179.595,6.463,149.059
C05315=1145.317,67.842,-52.257,-179.598,6.463,149.060
C05316=1145.323,67.592,-52.242,-179.601,6.461,149.060
C05317=1145.327,67.343,-52.225,-179.603,6.459,149.061
C05318=1145.333,67.093,-52.208,-179.605,6.459,149.061
C05319=1145.338,66.844,-52.191,-179.609,6.457,149.062
C05320=1145.342,66.594,-52.175,-179.611,6.456,149.062
C05321=1145.347,66.345,-52.159,-179.614,6.455,149.063
C05322=1145.352,66.096,-52.142,-179.617,6.454,149.064
C05323=1145.358,65.847,-52.126,-179.619,6.453,149.064
C05324=1145.363,65.596,-52.110,-179.622,6.451,149.064
C05325=1145.367,65.347,-52.093,-179.625,6.450,149.065
C05326=1145.372,65.098,-52.077,-179.627,6.449,149.066
C05327=1145.377,64.848,-52.061,-179.630,6.447,149.066
C05328=1145.382,64.599,-52.044,-179.632,6.447,149.067
C05329=1145.386,64.350,-52.028,-179.635,6.445,149.067
C05330=1145.393,64.100,-52.012,-179.638,6.443,149.067
C05331=1145.397,63.851,-51.995,-179.641,6.443,149.068
C05332=1145.402,63.601,-51.979,-179.643,6.441,149.069
C05333=1145.407,63.352,-51.963,-179.645,6.440,149.069
C05334=1145.412,63.103,-51.946,-179.649,6.439,149.070
C05335=1145.417,62.853,-51.930,-179.651,6.437,149.070
C05336=1145.422,62.604,-51.914,-179.654,6.437,149.071
C05337=1145.427,62.354,-51.898,-179.657,6.435,149.071
C05338=1145.432,62.105,-51.882,-179.659,6.434,149.072
C05339=1145.436,61.856,-51.865,-179.662,6.433,149.072
C05340=1145.442,61.606,-51.850,-179.664,6.432,149.073
C05341=1145.447,61.357,-51.832,-179.667,6.431,149.073
C05342=1145.452,61.107,-51.817,-179.670,6.429,149.074
C05343=1145.457,60.858,-51.800,-179.673,6.429,149.074
C05344=1145.462,60.608,-51.784,-179.675,6.427,149.075
C05345=1145.467,60.359,-51.768,-179.677,6.426,149.075
C05346=1145.472,60.109,-51.752,-179.681,6.425,149.076
C05347=1145.477,59.861,-51.736,-179.683,6.423,149.076
C05348=1145.482,59.610,-51.720,-179.686,6.422,149.077
C05349=1145.487,59.361,-51.704,-179.689,6.421,149.077
C05350=1145.492,59.112,-51.688,-179.691,6.420,149.078
C05351=1145.497,58.862,-51.672,-179.694,6.418,149.078
C05352=1145.502,58.613,-51.655,-179.696,6.418,149.079
C05353=1145.507,58.363,-51.640,-179.699,6.416,149.079
C05354=1145.511,58.114,-51.623,-179.701,6.416,149.080
C05355=1145.517,57.864,-51.608,-179.704,6.414,149.080
C05356=1145.522,57.615,-51.592,-179.707,6.413,149.081
C05357=1145.527,57.366,-51.575,-179.709,6.412,149.081
C05358=1145.531,57.116,-51.560,-179.713,6.410,149.082
C05359=1145.536,56.866,-51.544,-179.715,6.410,149.082
C05360=1145.541,56.618,-51.528,-179.718,6.408,149.083
C05361=1145.547,56.368,-51.512,-179.720,6.407,149.084
C05362=1145.551,56.118,-51.496,-179.723,6.406,149.084
C05363=1145.556,55.869,-51.480,-179.726,6.405,149.085
C05364=1145.562,55.620,-51.465,-179.728,6.404,149.085
C05365=1145.567,55.370,-51.449,-179.730,6.403,149.086
C05366=1145.572,55.121,-51.432,-179.734,6.402,149.086
C05367=1145.577,54.872,-51.417,-179.736,6.400,149.087
C05368=1145.582,54.621,-51.401,-179.739,6.399,149.087
C05369=1145.587,54.372,-51.386,-179.742,6.398,149.088
C05370=1145.591,54.123,-51.369,-179.744,6.397,149.088
C05371=1145.597,53.854,-51.352,-179.747,6.396,149.089
C05372=1145.602,53.586,-51.335,-179.750,6.394,149.089
C05373=1145.608,53.317,-51.319,-179.753,6.394,149.090
C05374=1145.614,53.048,-51.302,-179.755,6.392,149.090
C05375=1145.618,52.799,-51.285,-179.759,6.391,149.091
C05376=1145.623,52.549,-51.270,-179.761,6.390,149.092
C05377=1145.628,52.300,-51.255,-179.764,6.388,149.092
C05378=1145.633,52.051,-51.239,-179.766,6.388,149.093
C05379=1145.638,51.801,-51.223,-179.769,6.386,149.093
C05380=1145.644,51.551,-51.207,-179.771,6.385,149.094
C05381=1145.649,51.303,-51.191,-179.774,6.384,149.094
C05382=1145.653,51.053,-51.176,-179.776,6.383,149.095
C05383=1145.658,50.803,-51.160,-179.779,6.381,149.095
C05384=1145.663,50.554,-51.145,-179.782,6.381,149.096
C05385=1145.668,50.304,-51.129,-179.785,6.379,149.096
C05386=1145.673,50.055,-51.114,-179.787,6.379,149.097
C05387=1145.678,49.805,-51.098,-179.790,6.377,149.097
C05388=1145.684,49.556,-51.082,-179.792,6.376,149.098
C05389=1145.688,49.306,-51.067,-179.795,6.375,149.098
C05390=1145.693,49.057,-51.051,-179.798,6.374,149.099
C05391=1145.699,48.807,-51.036,-179.800,6.373,149.099
C05392=1145.704,48.558,-51.020,-179.803,6.372,149.100
C05393=1145.708,48.308,-51.005,-179.806,6.370,149.100
C05394=1145.713,48.059,-50.989,-179.808,6.370,149.101
C05395=1145.719,47.809,-50.974,-179.811,6.368,149.102
C05396=1145.723,47.560,-50.959,-179.813,6.368,149.102
C05397=1145.728,47.310,-50.943,-179.816,6.366,149.103
C05398=1145.734,47.061,-50.927,-179.819,6.365,149.103
C05399=1145.738,46.812,-50.912,-179.821,6.365,149.104
C05400=1145.744,46.562,-50.897,-179.824,6.363,149.104
C05401=1145.749,46.313,-50.881,-179.826,6.362,149.105
C05402=1145.753,46.063,-50.866,-179.829,6.361,149.105
C05403=1145.758,45.814,-50.850,-179.832,6.360,149.106
C05404=1145.764,45.564,-50.835,-179.834,6.359,149.106
C05405=1145.768,45.315,-50.820,-179.837,6.358,149.107
C05406=1145.774,45.066,-50.804,-179.840,6.357,149.107
C05407=1145.778,44.816,-50.789,-179.842,6.356,149.108
C05408=1145.783,44.567,-50.773,-179.845,6.354,149.108
C05409=1145.789,44.317,-50.758,-179.847,6.354,149.109
C05410=1145.794,44.068,-50.743,-179.851,6.352,149.110
C05411=1145.799,43.818,-50.728,-179.853,6.352,149.110
C05412=1145.804,43.569,-50.713,-179.855,6.350,149.110
C05413=1145.808,43.319,-50.697,-179.858,6.349,149.111
C05414=1145.813,43.070,-50.682,-179.860,6.349,149.112
C05415=1145.819,42.820,-50.667,-179.863,6.347,149.112
C05416=1145.824,42.570,-50.651,-179.866,6.346,149.113
C05417=1145.829,42.321,-50.636,-179.868,6.345,149.113
C05418=1145.834,42.072,-50.621,-179.871,6.344,149.114
C05419=1145.839,41.823,-50.606,-179.874,6.343,149.114
C05420=1145.844,41.572,-50.590,-179.876,6.342,149.115
C05421=1145.849,41.323,-50.575,-179.879,6.341,149.115
C05422=1145.854,41.074,-50.560,-179.881,6.340,149.116
C05423=1145.859,40.825,-50.545,-179.884,6.339,149.116
C05424=1145.864,40.575,-50.530,-179.887,6.338,149.117
C05425=1145.869,40.325,-50.515,-179.889,6.337,149.117
C05426=1145.874,40.076,-50.499,-179.892,6.336,149.118
C05427=1145.879,39.826,-50.485,-179.894,6.335,149.119
C05428=1145.885,39.577,-50.469,-179.898,6.333,149.119
C05429=1145.889,39.328,-50.454,-179.900,6.333,149.120
C05430=1145.894,39.077,-50.439,-179.902,6.332,149.120
C05431=1145.899,38.828,-50.424,-179.905,6.331,149.121
C05432=1145.904,38.579,-50.409,-179.907,6.330,149.121
C05433=1145.909,38.329,-50.394,-179.911,6.328,149.122
C05434=1145.914,38.080,-50.379,-179.913,6.328,149.122
C05435=1145.919,37.830,-50.364,-179.915,6.326,149.123
C05436=1145.924,37.581,-50.350,-179.918,6.325,149.123
C05437=1145.930,37.331,-50.334,-179.920,6.325,149.124
C05438=1145.935,37.082,-50.320,-179.924,6.323,149.125
C05439=1145.939,36.833,-50.305,-179.926,6.323,149.125
C05440=1145.945,36.583,-50.289,-179.928,6.321,149.125
C05441=1145.950,36.333,-50.275,-179.931,6.320,149.126
C05442=1145.955,36.084,-50.259,-179.933,6.320,149.127
C05443=1145.960,35.834,-50.245,-179.936,6.318,149.127
C05444=1145.965,35.585,-50.230,-179.939,6.318,149.128
C05445=1145.970,35.335,-50.215,-179.941,6.316,149.128
C05446=1145.975,35.086,-50.200,-179.944,6.315,149.129
C05447=1145.980,34.836,-50.186,-179.946,6.315,149.129
C05448=1145.985,34.587,-50.170,-179.949,6.313,149.130
C05449=1145.990,34.337,-50.156,-179.952,6.313,149.130
C05450=1145.995,34.088,-50.141,-179.954,6.311,149.131
C05451=1146.001,33.838,-50.126,-179.957,6.310,149.132
C05452=1146.005,33.589,-50.111,-179.959,6.310,149.132
C05453=1146.010,33.339,-50.097,-179.962,6.308,149.133
C05454=1146.016,33.090,-50.081,-179.965,6.307,149.133
C05455=1146.021,32.840,-50.067,-179.967,6.306,149.134
C05456=1146.026,32.591,-50.053,-179.970,6.305,149.134
C05457=1146.031,32.341,-50.037,-179.972,6.305,149.135
C05458=1146.036,32.091,-50.023,-179.975,6.303,149.135
C05459=1146.041,31.842,-50.008,-179.978,6.302,149.136
C05460=1146.046,31.593,-49.994,-179.980,6.302,149.136
C05461=1146.051,31.343,-49.979,-179.983,6.300,149.137
C05462=1146.056,31.093,-49.964,-179.985,6.300,149.137
C05463=1146.061,30.844,-49.949,-179.988,6.298,149.138
C05464=1146.066,30.595,-49.934,-179.991,6.297,149.139
C05465=1146.071,30.345,-49.920,-179.993,6.297,149.139
C05466=1146.077,30.096,-49.906,-179.996,6.295,149.140
C05467=1146.081,29.847,-49.891,-179.998,6.295,149.140
C05468=1146.086,29.597,-49.876,179.999,6.294,149.141
C05469=1146.091,29.347,-49.862,179.996,6.292,149.141
C05470=1146.097,29.098,-49.846,179.994,6.292,149.142
C05471=1146.102,28.848,-49.832,179.992,6.291,149.142
C05472=1146.107,28.598,-49.818,179.989,6.290,149.143
C05473=1146.112,28.349,-49.804,179.986,6.289,149.144
C05474=1146.116,28.100,-49.789,179.984,6.288,149.144
C05475=1146.122,27.830,-49.773,179.981,6.287,149.145
C05476=1146.128,27.561,-49.757,179.978,6.285,149.145
C05477=1146.133,27.293,-49.742,179.975,6.285,149.146
C05478=1146.138,27.024,-49.726,179.972,6.284,149.146
C05479=1146.144,26.774,-49.711,179.970,6.283,149.147
C05480=1146.149,26.524,-49.697,179.968,6.282,149.147
C05481=1146.154,26.275,-49.683,179.965,6.281,149.148
C05482=1146.159,26.025,-49.669,179.962,6.280,149.149
C05483=1146.164,25.775,-49.654,179.960,6.279,149.149
